LIN {X -0.197,Y -496.201,Z 1484.544,A 0.000,B 0.000,C 90.000,E1 97.936} C_DIS
LIN {X 0.122,Y -496.493,Z 1484.541,A 0.000,B 0.000,C 90.000,E1 97.409} C_DIS
LIN {X -0.111,Y -495.790,Z 1484.539,A 0.000,B 0.000,C 90.000,E1 96.947} C_DIS
LIN {X 0.150,Y -493.977,Z 1484.536,A 0.000,B 0.000,C 90.000,E1 96.429} C_DIS
LIN {X 0.006,Y -492.546,Z 1484.534,A 0.000,B 0.000,C 90.000,E1 96.201} C_DIS
LIN {X -0.163,Y -484.137,Z 1484.528,A 0.000,B 0.000,C 90.000,E1 94.992} C_DIS
LIN {X -0.014,Y -472.049,Z 1484.517,A 0.000,B 0.000,C 90.000,E1 92.980} C_DIS
LIN {X -0.036,Y -464.001,Z 1484.510,A 0.000,B 0.000,C 90.000,E1 91.718} C_DIS
LIN {X 0.053,Y -453.863,Z 1484.501,A 0.000,B 0.000,C 90.000,E1 90.172} C_DIS
LIN {X 0.159,Y -441.677,Z 1484.491,A 0.000,B 0.000,C 90.000,E1 88.339} C_DIS
LIN {X 0.042,Y -429.423,Z 1484.481,A 0.000,B 0.000,C 90.000,E1 86.502} C_DIS
LIN {X -0.173,Y -415.484,Z 1484.469,A 0.000,B 0.000,C 90.000,E1 84.375} C_DIS
LIN {X -0.004,Y -404.925,Z 1484.459,A 0.000,B 0.000,C 90.000,E1 82.704} C_DIS
LIN {X 0.094,Y -392.488,Z 1484.449,A 0.000,B 0.000,C 90.000,E1 80.735} C_DIS
LIN {X 0.042,Y -376.995,Z 1484.434,A 0.000,B 0.000,C 90.000,E1 78.173} C_DIS
LIN {X 0.185,Y -362.226,Z 1484.420,A 0.000,B 0.000,C 90.000,E1 75.519} C_DIS
LIN {X 0.053,Y -350.925,Z 1484.408,A 0.000,B 0.000,C 90.000,E1 73.449} C_DIS
LIN {X -0.007,Y -339.682,Z 1484.396,A 0.000,B 0.000,C 90.000,E1 71.329} C_DIS
LIN {X 0.011,Y -328.550,Z 1484.384,A 0.000,B 0.000,C 90.000,E1 69.156} C_DIS
LIN {X -0.003,Y -311.910,Z 1484.365,A 0.000,B 0.000,C 90.000,E1 65.665} C_DIS
LIN {X -0.046,Y -297.959,Z 1484.347,A 0.000,B 0.000,C 90.000,E1 62.410} C_DIS
LIN {X -0.061,Y -287.479,Z 1484.332,A 0.000,B 0.000,C 90.000,E1 59.744} C_DIS
LIN {X 0.186,Y -276.248,Z 1484.315,A 0.000,B 0.000,C 90.000,E1 56.628} C_DIS
LIN {X -0.025,Y -265.271,Z 1484.297,A 0.000,B 0.000,C 90.000,E1 53.543} C_DIS
LIN {X -0.025,Y -253.773,Z 1484.278,A 0.000,B 0.000,C 90.000,E1 49.989} C_DIS
LIN {X -0.097,Y -243.103,Z 1484.258,A 0.000,B 0.000,C 90.000,E1 46.377} C_DIS
LIN {X 0.079,Y -235.363,Z 1484.241,A 0.000,B 0.000,C 90.000,E1 43.380} C_DIS
LIN {X -0.020,Y -226.608,Z 1484.220,A 0.000,B 0.000,C 90.000,E1 39.644} C_DIS
LIN {X -0.002,Y -220.283,Z 1484.203,A 0.000,B 0.000,C 90.000,E1 36.583} C_DIS
LIN {X 0.007,Y -213.225,Z 1484.182,A 0.000,B 0.000,C 90.000,E1 32.704} C_DIS
LIN {X 0.105,Y -207.137,Z 1484.160,A 0.000,B 0.000,C 90.000,E1 28.743} C_DIS
LIN {X 0.059,Y -201.875,Z 1484.138,A 0.000,B 0.000,C 90.000,E1 24.771} C_DIS
LIN {X 0.031,Y -196.556,Z 1484.111,A 0.000,B 0.000,C 90.000,E1 19.939} C_DIS
LIN {X -0.035,Y -192.268,Z 1484.084,A 0.000,B 0.000,C 90.000,E1 15.064} C_DIS
LIN {X 0.082,Y -188.732,Z 1484.052,A 0.000,B 0.000,C 90.000,E1 9.265} C_DIS
LIN {X -0.046,Y -186.486,Z 1484.019,A 0.000,B 0.000,C 90.000,E1 3.498} C_DIS
LIN {X 0.034,Y -185.763,Z 1483.984,A 0.000,B 0.000,C 90.000,E1 357.020} C_DIS
LIN {X -0.001,Y -186.437,Z 1483.951,A 0.000,B 0.000,C 90.000,E1 351.197} C_DIS
LIN {X -0.087,Y -188.920,Z 1483.914,A 0.000,B 0.000,C 90.000,E1 344.574} C_DIS
LIN {X 0.063,Y -192.234,Z 1483.887,A 0.000,B 0.000,C 90.000,E1 339.571} C_DIS
LIN {X 0.014,Y -195.864,Z 1483.864,A 0.000,B 0.000,C 90.000,E1 335.485} C_DIS
LIN {X -0.045,Y -200.473,Z 1483.841,A 0.000,B 0.000,C 90.000,E1 331.435} C_DIS
LIN {X 0.084,Y -206.120,Z 1483.819,A 0.000,B 0.000,C 90.000,E1 327.375} C_DIS
LIN {X 0.075,Y -211.585,Z 1483.801,A 0.000,B 0.000,C 90.000,E1 324.196} C_DIS
LIN {X -0.068,Y -217.834,Z 1483.784,A 0.000,B 0.000,C 90.000,E1 321.090} C_DIS
LIN {X 0.048,Y -225.078,Z 1483.766,A 0.000,B 0.000,C 90.000,E1 317.957} C_DIS
LIN {X 0.113,Y -234.367,Z 1483.747,A 0.000,B 0.000,C 90.000,E1 314.514} C_DIS
LIN {X 0.146,Y -244.835,Z 1483.729,A 0.000,B 0.000,C 90.000,E1 311.148} C_DIS
LIN {X -0.015,Y -254.072,Z 1483.715,A 0.000,B 0.000,C 90.000,E1 308.624} C_DIS
LIN {X 0.023,Y -263.027,Z 1483.703,A 0.000,B 0.000,C 90.000,E1 306.457} C_DIS
LIN {X 0.002,Y -271.259,Z 1483.693,A 0.000,B 0.000,C 90.000,E1 304.692} C_DIS
LIN {X -0.041,Y -280.539,Z 1483.683,A 0.000,B 0.000,C 90.000,E1 302.959} C_DIS
LIN {X -0.120,Y -292.857,Z 1483.672,A 0.000,B 0.000,C 90.000,E1 300.924} C_DIS
LIN {X 0.122,Y -304.194,Z 1483.662,A 0.000,B 0.000,C 90.000,E1 299.205} C_DIS
LIN {X -0.090,Y -311.599,Z 1483.657,A 0.000,B 0.000,C 90.000,E1 298.281} C_DIS
LIN {X -0.012,Y -327.563,Z 1483.647,A 0.000,B 0.000,C 90.000,E1 296.437} C_DIS
LIN {X -0.040,Y -352.222,Z 1483.633,A 0.000,B 0.000,C 90.000,E1 293.898} C_DIS
LIN {X 0.157,Y -363.050,Z 1483.627,A 0.000,B 0.000,C 90.000,E1 292.770} C_DIS
LIN {X -0.133,Y -373.704,Z 1483.620,A 0.000,B 0.000,C 90.000,E1 291.716} C_DIS
LIN {X -0.119,Y -384.171,Z 1483.614,A 0.000,B 0.000,C 90.000,E1 290.610} C_DIS
LIN {X 0.094,Y -394.100,Z 1483.608,A 0.000,B 0.000,C 90.000,E1 289.504} C_DIS
LIN {X -0.132,Y -403.935,Z 1483.602,A 0.000,B 0.000,C 90.000,E1 288.417} C_DIS
LIN {X -0.156,Y -410.810,Z 1483.598,A 0.000,B 0.000,C 90.000,E1 287.583} C_DIS
LIN {X 0.001,Y -417.219,Z 1483.593,A 0.000,B 0.000,C 90.000,E1 286.732} C_DIS
LIN {X 0.104,Y -422.991,Z 1483.588,A 0.000,B 0.000,C 90.000,E1 285.898} C_DIS
LIN {X 0.144,Y -428.102,Z 1483.584,A 0.000,B 0.000,C 90.000,E1 285.079} C_DIS
LIN {X -0.066,Y -432.329,Z 1483.579,A 0.000,B 0.000,C 90.000,E1 284.300} C_DIS
LIN {X 0.069,Y -435.873,Z 1483.575,A 0.000,B 0.000,C 90.000,E1 283.480} C_DIS
LIN {X 0.139,Y -437.790,Z 1483.572,A 0.000,B 0.000,C 90.000,E1 282.939} C_DIS
LIN {X 0.114,Y -439.351,Z 1483.569,A 0.000,B 0.000,C 90.000,E1 282.411} C_DIS
LIN {X 0.100,Y -440.535,Z 1483.566,A 0.000,B 0.000,C 90.000,E1 281.883} C_DIS
LIN {X 0.006,Y -441.261,Z 1483.563,A 0.000,B 0.000,C 90.000,E1 281.366} C_DIS
LIN {X 0.009,Y -441.485,Z 1483.560,A 0.000,B 0.000,C 90.000,E1 280.838} C_DIS
LIN {X 0.015,Y -441.181,Z 1483.557,A 0.000,B 0.000,C 90.000,E1 280.310} C_DIS
LIN {X -0.057,Y -440.296,Z 1483.554,A 0.000,B 0.000,C 90.000,E1 279.792} C_DIS
LIN {X -0.054,Y -438.823,Z 1483.551,A 0.000,B 0.000,C 90.000,E1 279.265} C_DIS
LIN {X -0.128,Y -436.665,Z 1483.548,A 0.000,B 0.000,C 90.000,E1 278.746} C_DIS
LIN {X -0.144,Y -433.693,Z 1483.546,A 0.000,B 0.000,C 90.000,E1 278.219} C_DIS
LIN {X 0.184,Y -429.791,Z 1483.543,A 0.000,B 0.000,C 90.000,E1 277.644} C_DIS
LIN {X 0.066,Y -424.843,Z 1483.540,A 0.000,B 0.000,C 90.000,E1 277.125} C_DIS
LIN {X 0.036,Y -418.911,Z 1483.537,A 0.000,B 0.000,C 90.000,E1 276.606} C_DIS
LIN {X 0.027,Y -412.593,Z 1483.534,A 0.000,B 0.000,C 90.000,E1 276.144} C_DIS
LIN {X 0.065,Y -406.271,Z 1483.532,A 0.000,B 0.000,C 90.000,E1 275.739} C_DIS
LIN {X -0.003,Y -399.690,Z 1483.530,A 0.000,B 0.000,C 90.000,E1 275.391} C_DIS
LIN {X 0.013,Y -389.854,Z 1483.527,A 0.000,B 0.000,C 90.000,E1 274.935} C_DIS
LIN {X -0.072,Y -374.378,Z 1483.524,A 0.000,B 0.000,C 90.000,E1 274.302} C_DIS
LIN {X 0.041,Y -361.581,Z 1483.521,A 0.000,B 0.000,C 90.000,E1 273.784} C_DIS
LIN {X 0.034,Y -348.652,Z 1483.519,A 0.000,B 0.000,C 90.000,E1 273.326} C_DIS
LIN {X -0.080,Y -338.477,Z 1483.517,A 0.000,B 0.000,C 90.000,E1 273.037} C_DIS
LIN {X -0.048,Y -324.878,Z 1483.515,A 0.000,B 0.000,C 90.000,E1 272.694} C_DIS
LIN {X 0.022,Y -313.880,Z 1483.514,A 0.000,B 0.000,C 90.000,E1 272.465} C_DIS
LIN {X -0.011,Y -300.345,Z 1483.513,A 0.000,B 0.000,C 90.000,E1 272.293} C_DIS
LIN {X -0.077,Y -289.823,Z 1483.512,A 0.000,B 0.000,C 90.000,E1 272.236} C_DIS
LIN {X -0.124,Y -286.503,Z 1483.512,A 0.000,B 0.000,C 90.000,E1 272.236} C_DIS
LIN {X 0.072,Y -181.230,Z 1483.512,A 0.000,B 0.000,C 90.000,E1 272.178} C_DIS
LIN {X 0.063,Y -181.568,Z 1483.503,A 0.000,B 0.000,C 90.000,E1 270.458} C_DIS
LIN {X 0.053,Y -181.117,Z 1483.489,A 0.000,B 0.000,C 90.000,E1 267.936} C_DIS
LIN {X 0.041,Y -180.906,Z 1483.475,A 0.000,B 0.000,C 90.000,E1 265.412} C_DIS
LIN {X -0.083,Y -180.716,Z 1483.470,A 0.000,B 0.000,C 90.000,E1 264.609} C_DIS
LIN {X 0.015,Y -178.803,Z 1483.442,A 0.000,B 0.000,C 90.000,E1 259.511} C_DIS
LIN {X 0.091,Y -175.849,Z 1483.413,A 0.000,B 0.000,C 90.000,E1 254.393} C_DIS
LIN {X 0.051,Y -172.584,Z 1483.390,A 0.000,B 0.000,C 90.000,E1 250.134} C_DIS
LIN {X 0.067,Y -171.473,Z 1483.380,A 0.000,B 0.000,C 90.000,E1 248.411} C_DIS
LIN {X 0.047,Y -167.704,Z 1483.356,A 0.000,B 0.000,C 90.000,E1 244.101} C_DIS
LIN {X 0.060,Y -166.390,Z 1483.347,A 0.000,B 0.000,C 90.000,E1 242.359} C_DIS
LIN {X 0.051,Y -163.117,Z 1483.327,A 0.000,B 0.000,C 90.000,E1 238.869} C_DIS
LIN {X 0.101,Y -161.067,Z 1483.313,A 0.000,B 0.000,C 90.000,E1 236.215} C_DIS
LIN {X -0.012,Y -157.800,Z 1483.293,A 0.000,B 0.000,C 90.000,E1 232.718} C_DIS
LIN {X -0.073,Y -155.836,Z 1483.278,A 0.000,B 0.000,C 90.000,E1 230.070} C_DIS
LIN {X -0.017,Y -152.086,Z 1483.253,A 0.000,B 0.000,C 90.000,E1 225.567} C_DIS
LIN {X 0.002,Y -150.336,Z 1483.238,A 0.000,B 0.000,C 90.000,E1 222.852} C_DIS
LIN {X 0.023,Y -147.076,Z 1483.213,A 0.000,B 0.000,C 90.000,E1 218.302} C_DIS
LIN {X -0.073,Y -145.650,Z 1483.198,A 0.000,B 0.000,C 90.000,E1 215.598} C_DIS
LIN {X -0.068,Y -143.032,Z 1483.172,A 0.000,B 0.000,C 90.000,E1 211.003} C_DIS
LIN {X 0.058,Y -141.657,Z 1483.152,A 0.000,B 0.000,C 90.000,E1 207.257} C_DIS
LIN {X -0.023,Y -139.446,Z 1483.115,A 0.000,B 0.000,C 90.000,E1 200.791} C_DIS
LIN {X 0.030,Y -139.180,Z 1483.105,A 0.000,B 0.000,C 90.000,E1 198.906} C_DIS
LIN {X 0.058,Y -138.320,Z 1483.053,A 0.000,B 0.000,C 90.000,E1 189.557} C_DIS
LIN {X 0.067,Y -139.465,Z 1483.006,A 0.000,B 0.000,C 90.000,E1 181.146} C_DIS
LIN {X 0.009,Y -141.029,Z 1482.975,A 0.000,B 0.000,C 90.000,E1 175.584} C_DIS
LIN {X -0.037,Y -142.396,Z 1482.960,A 0.000,B 0.000,C 90.000,E1 172.818} C_DIS
LIN {X 0.025,Y -144.628,Z 1482.934,A 0.000,B 0.000,C 90.000,E1 168.173} C_DIS
LIN {X -0.057,Y -147.823,Z 1482.909,A 0.000,B 0.000,C 90.000,E1 163.614} C_DIS
LIN {X 0.031,Y -150.514,Z 1482.889,A 0.000,B 0.000,C 90.000,E1 159.934} C_DIS
LIN {X 0.050,Y -153.976,Z 1482.868,A 0.000,B 0.000,C 90.000,E1 156.305} C_DIS
LIN {X -0.028,Y -157.388,Z 1482.849,A 0.000,B 0.000,C 90.000,E1 152.743} C_DIS
LIN {X -0.087,Y -161.592,Z 1482.829,A 0.000,B 0.000,C 90.000,E1 149.203} C_DIS
LIN {X -0.076,Y -165.788,Z 1482.809,A 0.000,B 0.000,C 90.000,E1 145.674} C_DIS
LIN {X -0.091,Y -170.751,Z 1482.790,A 0.000,B 0.000,C 90.000,E1 142.190} C_DIS
LIN {X 0.067,Y -175.623,Z 1482.771,A 0.000,B 0.000,C 90.000,E1 138.690} C_DIS
LIN {X -0.063,Y -181.239,Z 1482.752,A 0.000,B 0.000,C 90.000,E1 135.324} C_DIS
LIN {X 0.067,Y -186.708,Z 1482.733,A 0.000,B 0.000,C 90.000,E1 131.919} C_DIS
LIN {X 0.019,Y -191.308,Z 1482.719,A 0.000,B 0.000,C 90.000,E1 129.439} C_DIS
LIN {X -0.050,Y -197.137,Z 1482.701,A 0.000,B 0.000,C 90.000,E1 126.171} C_DIS
LIN {X -0.035,Y -201.174,Z 1482.689,A 0.000,B 0.000,C 90.000,E1 124.119} C_DIS
LIN {X -0.001,Y -201.373,Z 1482.689,A 0.000,B 0.000,C 90.000,E1 123.992} C_DIS
LIN {X -0.046,Y -314.503,Z 1482.689,A 0.000,B 0.000,C 90.000,E1 123.992} C_DIS
LIN {X -0.172,Y -315.934,Z 1482.689,A 0.000,B 0.000,C 90.000,E1 123.992} C_DIS
LIN {X 0.069,Y -321.100,Z 1482.687,A 0.000,B 0.000,C 90.000,E1 123.706} C_DIS
LIN {X 0.043,Y -324.274,Z 1482.686,A 0.000,B 0.000,C 90.000,E1 123.420} C_DIS
LIN {X 0.155,Y -327.904,Z 1482.683,A 0.000,B 0.000,C 90.000,E1 122.880} C_DIS
LIN {X -0.025,Y -329.447,Z 1482.681,A 0.000,B 0.000,C 90.000,E1 122.594} C_DIS
LIN {X 0.010,Y -342.874,Z 1482.662,A 0.000,B 0.000,C 90.000,E1 119.155} C_DIS
LIN {X -0.017,Y -355.319,Z 1482.647,A 0.000,B 0.000,C 90.000,E1 116.411} C_DIS
LIN {X 0.144,Y -369.261,Z 1482.632,A 0.000,B 0.000,C 90.000,E1 113.695} C_DIS
LIN {X -0.205,Y -383.004,Z 1482.619,A 0.000,B 0.000,C 90.000,E1 111.408} C_DIS
LIN {X 0.007,Y -398.116,Z 1482.606,A 0.000,B 0.000,C 90.000,E1 109.087} C_DIS
LIN {X -0.036,Y -414.704,Z 1482.594,A 0.000,B 0.000,C 90.000,E1 106.858} C_DIS
LIN {X 0.100,Y -432.882,Z 1482.582,A 0.000,B 0.000,C 90.000,E1 104.662} C_DIS
LIN {X -0.096,Y -452.544,Z 1482.570,A 0.000,B 0.000,C 90.000,E1 102.591} C_DIS
LIN {X -0.093,Y -472.851,Z 1482.559,A 0.000,B 0.000,C 90.000,E1 100.658} C_DIS
LIN {X -0.172,Y -488.418,Z 1482.552,A 0.000,B 0.000,C 90.000,E1 99.321} C_DIS
LIN {X -0.094,Y -490.656,Z 1482.550,A 0.000,B 0.000,C 90.000,E1 99.095} C_DIS
LIN {X 0.061,Y -492.347,Z 1482.549,A 0.000,B 0.000,C 90.000,E1 98.859} C_DIS
LIN {X -0.034,Y -493.807,Z 1482.548,A 0.000,B 0.000,C 90.000,E1 98.624} C_DIS
LIN {X -0.202,Y -494.892,Z 1482.547,A 0.000,B 0.000,C 90.000,E1 98.398} C_DIS
LIN {X 0.114,Y -496.149,Z 1482.544,A 0.000,B 0.000,C 90.000,E1 97.871} C_DIS
LIN {X -0.127,Y -496.370,Z 1482.541,A 0.000,B 0.000,C 90.000,E1 97.409} C_DIS
LIN {X 0.132,Y -495.595,Z 1482.538,A 0.000,B 0.000,C 90.000,E1 96.891} C_DIS
LIN {X -0.099,Y -493.693,Z 1482.536,A 0.000,B 0.000,C 90.000,E1 96.429} C_DIS
LIN {X -0.242,Y -492.203,Z 1482.534,A 0.000,B 0.000,C 90.000,E1 96.201} C_DIS
LIN {X 0.070,Y -483.811,Z 1482.527,A 0.000,B 0.000,C 90.000,E1 94.935} C_DIS
LIN {X 0.207,Y -471.696,Z 1482.516,A 0.000,B 0.000,C 90.000,E1 92.922} C_DIS
LIN {X 0.177,Y -463.645,Z 1482.509,A 0.000,B 0.000,C 90.000,E1 91.661} C_DIS
LIN {X -0.197,Y -453.496,Z 1482.501,A 0.000,B 0.000,C 90.000,E1 90.172} C_DIS
LIN {X 0.101,Y -439.614,Z 1482.489,A 0.000,B 0.000,C 90.000,E1 88.051} C_DIS
LIN {X -0.067,Y -427.391,Z 1482.479,A 0.000,B 0.000,C 90.000,E1 86.216} C_DIS
LIN {X -0.008,Y -415.232,Z 1482.468,A 0.000,B 0.000,C 90.000,E1 84.318} C_DIS
LIN {X 0.152,Y -404.703,Z 1482.459,A 0.000,B 0.000,C 90.000,E1 82.648} C_DIS
LIN {X -0.150,Y -392.292,Z 1482.448,A 0.000,B 0.000,C 90.000,E1 80.735} C_DIS
LIN {X -0.198,Y -376.851,Z 1482.434,A 0.000,B 0.000,C 90.000,E1 78.173} C_DIS
LIN {X -0.048,Y -362.083,Z 1482.420,A 0.000,B 0.000,C 90.000,E1 75.519} C_DIS
LIN {X -0.077,Y -350.793,Z 1482.408,A 0.000,B 0.000,C 90.000,E1 73.433} C_DIS
LIN {X 0.090,Y -339.540,Z 1482.396,A 0.000,B 0.000,C 90.000,E1 71.275} C_DIS
LIN {X -0.092,Y -328.391,Z 1482.384,A 0.000,B 0.000,C 90.000,E1 69.135} C_DIS
LIN {X 0.067,Y -311.746,Z 1482.365,A 0.000,B 0.000,C 90.000,E1 65.613} C_DIS
LIN {X 0.009,Y -297.800,Z 1482.346,A 0.000,B 0.000,C 90.000,E1 62.359} C_DIS
LIN {X 0.107,Y -286.054,Z 1482.330,A 0.000,B 0.000,C 90.000,E1 59.331} C_DIS
LIN {X -0.015,Y -276.142,Z 1482.315,A 0.000,B 0.000,C 90.000,E1 56.628} C_DIS
LIN {X 0.076,Y -266.397,Z 1482.299,A 0.000,B 0.000,C 90.000,E1 53.829} C_DIS
LIN {X 0.107,Y -254.835,Z 1482.279,A 0.000,B 0.000,C 90.000,E1 50.275} C_DIS
LIN {X -0.104,Y -245.127,Z 1482.261,A 0.000,B 0.000,C 90.000,E1 47.067} C_DIS
LIN {X -0.040,Y -237.225,Z 1482.245,A 0.000,B 0.000,C 90.000,E1 44.109} C_DIS
LIN {X -0.097,Y -228.340,Z 1482.224,A 0.000,B 0.000,C 90.000,E1 40.378} C_DIS
LIN {X -0.035,Y -221.856,Z 1482.207,A 0.000,B 0.000,C 90.000,E1 37.317} C_DIS
LIN {X -0.028,Y -214.705,Z 1482.186,A 0.000,B 0.000,C 90.000,E1 33.452} C_DIS
LIN {X -0.060,Y -208.438,Z 1482.164,A 0.000,B 0.000,C 90.000,E1 29.539} C_DIS
LIN {X 0.033,Y -203.062,Z 1482.142,A 0.000,B 0.000,C 90.000,E1 25.540} C_DIS
LIN {X -0.018,Y -198.447,Z 1482.120,A 0.000,B 0.000,C 90.000,E1 21.535} C_DIS
LIN {X -0.074,Y -193.824,Z 1482.093,A 0.000,B 0.000,C 90.000,E1 16.677} C_DIS
LIN {X 0.063,Y -190.333,Z 1482.065,A 0.000,B 0.000,C 90.000,E1 11.715} C_DIS
LIN {X -0.067,Y -187.547,Z 1482.033,A 0.000,B 0.000,C 90.000,E1 5.967} C_DIS
LIN {X 0.051,Y -186.066,Z 1481.993,A 0.000,B 0.000,C 90.000,E1 358.682} C_DIS
LIN {X -0.026,Y -186.346,Z 1481.960,A 0.000,B 0.000,C 90.000,E1 352.875} C_DIS
LIN {X -0.054,Y -187.991,Z 1481.928,A 0.000,B 0.000,C 90.000,E1 347.061} C_DIS
LIN {X -0.087,Y -191.206,Z 1481.896,A 0.000,B 0.000,C 90.000,E1 341.275} C_DIS
LIN {X 0.047,Y -195.244,Z 1481.868,A 0.000,B 0.000,C 90.000,E1 336.305} C_DIS
LIN {X 0.054,Y -199.627,Z 1481.846,A 0.000,B 0.000,C 90.000,E1 332.231} C_DIS
LIN {X 0.048,Y -205.025,Z 1481.823,A 0.000,B 0.000,C 90.000,E1 328.201} C_DIS
LIN {X 0.008,Y -210.284,Z 1481.806,A 0.000,B 0.000,C 90.000,E1 325.022} C_DIS
LIN {X -0.124,Y -216.327,Z 1481.788,A 0.000,B 0.000,C 90.000,E1 321.904} C_DIS
LIN {X -0.048,Y -223.331,Z 1481.771,A 0.000,B 0.000,C 90.000,E1 318.771} C_DIS
LIN {X -0.141,Y -231.303,Z 1481.754,A 0.000,B 0.000,C 90.000,E1 315.729} C_DIS
LIN {X -0.039,Y -241.369,Z 1481.735,A 0.000,B 0.000,C 90.000,E1 312.324} C_DIS
LIN {X 0.035,Y -248.831,Z 1481.723,A 0.000,B 0.000,C 90.000,E1 310.092} C_DIS
LIN {X -0.076,Y -257.124,Z 1481.711,A 0.000,B 0.000,C 90.000,E1 307.935} C_DIS
LIN {X -0.145,Y -266.383,Z 1481.699,A 0.000,B 0.000,C 90.000,E1 305.804} C_DIS
LIN {X 0.029,Y -273.154,Z 1481.691,A 0.000,B 0.000,C 90.000,E1 304.358} C_DIS
LIN {X 0.015,Y -282.589,Z 1481.681,A 0.000,B 0.000,C 90.000,E1 302.625} C_DIS
LIN {X -0.028,Y -297.247,Z 1481.668,A 0.000,B 0.000,C 90.000,E1 300.256} C_DIS
LIN {X -0.115,Y -306.561,Z 1481.661,A 0.000,B 0.000,C 90.000,E1 298.949} C_DIS
LIN {X -0.135,Y -314.339,Z 1481.655,A 0.000,B 0.000,C 90.000,E1 297.975} C_DIS
LIN {X -0.015,Y -333.246,Z 1481.644,A 0.000,B 0.000,C 90.000,E1 295.848} C_DIS
LIN {X 0.040,Y -352.274,Z 1481.633,A 0.000,B 0.000,C 90.000,E1 293.898} C_DIS
LIN {X -0.009,Y -362.988,Z 1481.627,A 0.000,B 0.000,C 90.000,E1 292.823} C_DIS
LIN {X -0.075,Y -376.275,Z 1481.619,A 0.000,B 0.000,C 90.000,E1 291.461} C_DIS
LIN {X 0.064,Y -389.204,Z 1481.612,A 0.000,B 0.000,C 90.000,E1 290.066} C_DIS
LIN {X 0.163,Y -396.749,Z 1481.607,A 0.000,B 0.000,C 90.000,E1 289.214} C_DIS
LIN {X -0.042,Y -406.456,Z 1481.601,A 0.000,B 0.000,C 90.000,E1 288.127} C_DIS
LIN {X 0.085,Y -413.192,Z 1481.596,A 0.000,B 0.000,C 90.000,E1 287.275} C_DIS
LIN {X 0.153,Y -419.463,Z 1481.591,A 0.000,B 0.000,C 90.000,E1 286.441} C_DIS
LIN {X -0.135,Y -425.055,Z 1481.587,A 0.000,B 0.000,C 90.000,E1 285.662} C_DIS
LIN {X -0.239,Y -428.397,Z 1481.584,A 0.000,B 0.000,C 90.000,E1 285.134} C_DIS
LIN {X -0.031,Y -432.655,Z 1481.579,A 0.000,B 0.000,C 90.000,E1 284.300} C_DIS
LIN {X 0.107,Y -436.190,Z 1481.575,A 0.000,B 0.000,C 90.000,E1 283.480} C_DIS
LIN {X 0.179,Y -438.099,Z 1481.572,A 0.000,B 0.000,C 90.000,E1 282.939} C_DIS
LIN {X 0.155,Y -439.678,Z 1481.569,A 0.000,B 0.000,C 90.000,E1 282.411} C_DIS
LIN {X 0.142,Y -440.886,Z 1481.566,A 0.000,B 0.000,C 90.000,E1 281.883} C_DIS
LIN {X 0.052,Y -441.623,Z 1481.563,A 0.000,B 0.000,C 90.000,E1 281.366} C_DIS
LIN {X 0.057,Y -441.885,Z 1481.560,A 0.000,B 0.000,C 90.000,E1 280.838} C_DIS
LIN {X 0.064,Y -441.638,Z 1481.557,A 0.000,B 0.000,C 90.000,E1 280.310} C_DIS
LIN {X -0.006,Y -440.799,Z 1481.554,A 0.000,B 0.000,C 90.000,E1 279.792} C_DIS
LIN {X 0.000,Y -439.363,Z 1481.552,A 0.000,B 0.000,C 90.000,E1 279.265} C_DIS
LIN {X -0.072,Y -437.236,Z 1481.549,A 0.000,B 0.000,C 90.000,E1 278.746} C_DIS
LIN {X -0.085,Y -434.334,Z 1481.546,A 0.000,B 0.000,C 90.000,E1 278.219} C_DIS
LIN {X -0.180,Y -430.506,Z 1481.543,A 0.000,B 0.000,C 90.000,E1 277.701} C_DIS
LIN {X 0.132,Y -425.600,Z 1481.540,A 0.000,B 0.000,C 90.000,E1 277.125} C_DIS
LIN {X 0.081,Y -419.682,Z 1481.537,A 0.000,B 0.000,C 90.000,E1 276.606} C_DIS
LIN {X 0.103,Y -413.484,Z 1481.534,A 0.000,B 0.000,C 90.000,E1 276.144} C_DIS
LIN {X 0.096,Y -407.116,Z 1481.532,A 0.000,B 0.000,C 90.000,E1 275.739} C_DIS
LIN {X 0.031,Y -400.572,Z 1481.530,A 0.000,B 0.000,C 90.000,E1 275.391} C_DIS
LIN {X 0.031,Y -390.740,Z 1481.527,A 0.000,B 0.000,C 90.000,E1 274.935} C_DIS
LIN {X -0.099,Y -375.021,Z 1481.524,A 0.000,B 0.000,C 90.000,E1 274.302} C_DIS
LIN {X 0.016,Y -362.205,Z 1481.521,A 0.000,B 0.000,C 90.000,E1 273.784} C_DIS
LIN {X -0.011,Y -352.505,Z 1481.519,A 0.000,B 0.000,C 90.000,E1 273.440} C_DIS
LIN {X 0.132,Y -342.469,Z 1481.517,A 0.000,B 0.000,C 90.000,E1 273.094} C_DIS
LIN {X 0.022,Y -328.689,Z 1481.515,A 0.000,B 0.000,C 90.000,E1 272.751} C_DIS
LIN {X 0.045,Y -317.797,Z 1481.514,A 0.000,B 0.000,C 90.000,E1 272.522} C_DIS
LIN {X -0.046,Y -310.093,Z 1481.513,A 0.000,B 0.000,C 90.000,E1 272.407} C_DIS
LIN {X 0.128,Y -297.244,Z 1481.513,A 0.000,B 0.000,C 90.000,E1 272.236} C_DIS
LIN {X -0.099,Y -287.867,Z 1481.512,A 0.000,B 0.000,C 90.000,E1 272.236} C_DIS
LIN {X 0.088,Y -181.229,Z 1481.512,A 0.000,B 0.000,C 90.000,E1 272.178} C_DIS
LIN {X 0.049,Y -181.568,Z 1481.503,A 0.000,B 0.000,C 90.000,E1 270.458} C_DIS
LIN {X -0.091,Y -181.003,Z 1481.484,A 0.000,B 0.000,C 90.000,E1 267.135} C_DIS
LIN {X 0.026,Y -180.907,Z 1481.475,A 0.000,B 0.000,C 90.000,E1 265.412} C_DIS
LIN {X -0.098,Y -180.714,Z 1481.470,A 0.000,B 0.000,C 90.000,E1 264.609} C_DIS
LIN {X 0.001,Y -178.801,Z 1481.442,A 0.000,B 0.000,C 90.000,E1 259.511} C_DIS
LIN {X 0.078,Y -175.846,Z 1481.413,A 0.000,B 0.000,C 90.000,E1 254.393} C_DIS
LIN {X 0.077,Y -172.038,Z 1481.385,A 0.000,B 0.000,C 90.000,E1 249.263} C_DIS
LIN {X 0.053,Y -171.469,Z 1481.380,A 0.000,B 0.000,C 90.000,E1 248.411} C_DIS
LIN {X 0.033,Y -167.701,Z 1481.356,A 0.000,B 0.000,C 90.000,E1 244.101} C_DIS
LIN {X 0.046,Y -166.386,Z 1481.347,A 0.000,B 0.000,C 90.000,E1 242.359} C_DIS
LIN {X 0.038,Y -163.113,Z 1481.327,A 0.000,B 0.000,C 90.000,E1 238.869} C_DIS
LIN {X 0.088,Y -161.062,Z 1481.313,A 0.000,B 0.000,C 90.000,E1 236.215} C_DIS
LIN {X -0.025,Y -157.796,Z 1481.293,A 0.000,B 0.000,C 90.000,E1 232.718} C_DIS
LIN {X 0.014,Y -155.832,Z 1481.278,A 0.000,B 0.000,C 90.000,E1 230.033} C_DIS
LIN {X -0.029,Y -152.083,Z 1481.253,A 0.000,B 0.000,C 90.000,E1 225.567} C_DIS
LIN {X -0.010,Y -150.333,Z 1481.238,A 0.000,B 0.000,C 90.000,E1 222.852} C_DIS
LIN {X 0.010,Y -147.073,Z 1481.213,A 0.000,B 0.000,C 90.000,E1 218.302} C_DIS
LIN {X -0.086,Y -145.647,Z 1481.198,A 0.000,B 0.000,C 90.000,E1 215.598} C_DIS
LIN {X -0.081,Y -143.030,Z 1481.172,A 0.000,B 0.000,C 90.000,E1 211.003} C_DIS
LIN {X 0.046,Y -141.655,Z 1481.151,A 0.000,B 0.000,C 90.000,E1 207.257} C_DIS
LIN {X -0.035,Y -139.445,Z 1481.115,A 0.000,B 0.000,C 90.000,E1 200.791} C_DIS
LIN {X 0.017,Y -139.179,Z 1481.105,A 0.000,B 0.000,C 90.000,E1 198.906} C_DIS
LIN {X 0.046,Y -138.320,Z 1481.053,A 0.000,B 0.000,C 90.000,E1 189.557} C_DIS
LIN {X 0.055,Y -139.467,Z 1481.006,A 0.000,B 0.000,C 90.000,E1 181.146} C_DIS
LIN {X -0.004,Y -141.032,Z 1480.975,A 0.000,B 0.000,C 90.000,E1 175.584} C_DIS
LIN {X -0.050,Y -142.398,Z 1480.960,A 0.000,B 0.000,C 90.000,E1 172.818} C_DIS
LIN {X 0.013,Y -144.631,Z 1480.934,A 0.000,B 0.000,C 90.000,E1 168.173} C_DIS
LIN {X 0.074,Y -147.826,Z 1480.909,A 0.000,B 0.000,C 90.000,E1 163.559} C_DIS
LIN {X 0.017,Y -150.519,Z 1480.889,A 0.000,B 0.000,C 90.000,E1 159.934} C_DIS
LIN {X 0.038,Y -153.981,Z 1480.868,A 0.000,B 0.000,C 90.000,E1 156.305} C_DIS
LIN {X -0.042,Y -157.393,Z 1480.849,A 0.000,B 0.000,C 90.000,E1 152.743} C_DIS
LIN {X 0.039,Y -161.598,Z 1480.829,A 0.000,B 0.000,C 90.000,E1 149.154} C_DIS
LIN {X -0.089,Y -165.795,Z 1480.809,A 0.000,B 0.000,C 90.000,E1 145.674} C_DIS
LIN {X 0.031,Y -170.758,Z 1480.790,A 0.000,B 0.000,C 90.000,E1 142.145} C_DIS
LIN {X 0.053,Y -175.630,Z 1480.771,A 0.000,B 0.000,C 90.000,E1 138.690} C_DIS
LIN {X -0.078,Y -181.245,Z 1480.752,A 0.000,B 0.000,C 90.000,E1 135.324} C_DIS
LIN {X 0.053,Y -186.716,Z 1480.733,A 0.000,B 0.000,C 90.000,E1 131.919} C_DIS
LIN {X 0.004,Y -191.315,Z 1480.719,A 0.000,B 0.000,C 90.000,E1 129.439} C_DIS
LIN {X -0.065,Y -197.146,Z 1480.701,A 0.000,B 0.000,C 90.000,E1 126.171} C_DIS
LIN {X -0.048,Y -201.180,Z 1480.689,A 0.000,B 0.000,C 90.000,E1 124.119} C_DIS
LIN {X -0.059,Y -201.320,Z 1480.689,A 0.000,B 0.000,C 90.000,E1 124.040} C_DIS
LIN {X 0.120,Y -314.129,Z 1480.689,A 0.000,B 0.000,C 90.000,E1 123.992} C_DIS
LIN {X -0.022,Y -315.844,Z 1480.689,A 0.000,B 0.000,C 90.000,E1 123.992} C_DIS
LIN {X 0.045,Y -321.408,Z 1480.687,A 0.000,B 0.000,C 90.000,E1 123.706} C_DIS
LIN {X -0.057,Y -324.547,Z 1480.686,A 0.000,B 0.000,C 90.000,E1 123.420} C_DIS
LIN {X -0.078,Y -328.148,Z 1480.683,A 0.000,B 0.000,C 90.000,E1 122.880} C_DIS
LIN {X 0.020,Y -329.610,Z 1480.681,A 0.000,B 0.000,C 90.000,E1 122.546} C_DIS
LIN {X 0.090,Y -341.721,Z 1480.663,A 0.000,B 0.000,C 90.000,E1 119.411} C_DIS
LIN {X 0.026,Y -354.030,Z 1480.648,A 0.000,B 0.000,C 90.000,E1 116.668} C_DIS
LIN {X 0.158,Y -367.818,Z 1480.633,A 0.000,B 0.000,C 90.000,E1 113.951} C_DIS
LIN {X -0.081,Y -381.417,Z 1480.620,A 0.000,B 0.000,C 90.000,E1 111.642} C_DIS
LIN {X 0.088,Y -396.374,Z 1480.607,A 0.000,B 0.000,C 90.000,E1 109.322} C_DIS
LIN {X 0.000,Y -412.795,Z 1480.595,A 0.000,B 0.000,C 90.000,E1 107.094} C_DIS
LIN {X 0.085,Y -430.794,Z 1480.583,A 0.000,B 0.000,C 90.000,E1 104.898} C_DIS
LIN {X -0.211,Y -450.327,Z 1480.571,A 0.000,B 0.000,C 90.000,E1 102.827} C_DIS
LIN {X 0.102,Y -470.575,Z 1480.560,A 0.000,B 0.000,C 90.000,E1 100.838} C_DIS
LIN {X 0.068,Y -488.718,Z 1480.552,A 0.000,B 0.000,C 90.000,E1 99.265} C_DIS
LIN {X 0.213,Y -490.861,Z 1480.550,A 0.000,B 0.000,C 90.000,E1 99.029} C_DIS
LIN {X -0.205,Y -492.489,Z 1480.549,A 0.000,B 0.000,C 90.000,E1 98.859} C_DIS
LIN {X 0.189,Y -493.887,Z 1480.548,A 0.000,B 0.000,C 90.000,E1 98.568} C_DIS
LIN {X 0.021,Y -494.919,Z 1480.546,A 0.000,B 0.000,C 90.000,E1 98.341} C_DIS
LIN {X -0.153,Y -496.094,Z 1480.544,A 0.000,B 0.000,C 90.000,E1 97.871} C_DIS
LIN {X 0.098,Y -496.241,Z 1480.541,A 0.000,B 0.000,C 90.000,E1 97.352} C_DIS
LIN {X -0.134,Y -495.388,Z 1480.538,A 0.000,B 0.000,C 90.000,E1 96.891} C_DIS
LIN {X 0.125,Y -493.391,Z 1480.536,A 0.000,B 0.000,C 90.000,E1 96.372} C_DIS
LIN {X -0.111,Y -490.091,Z 1480.533,A 0.000,B 0.000,C 90.000,E1 95.910} C_DIS
LIN {X -0.005,Y -480.369,Z 1480.525,A 0.000,B 0.000,C 90.000,E1 94.416} C_DIS
LIN {X -0.060,Y -471.341,Z 1480.516,A 0.000,B 0.000,C 90.000,E1 92.922} C_DIS
LIN {X 0.100,Y -464.933,Z 1480.511,A 0.000,B 0.000,C 90.000,E1 91.892} C_DIS
LIN {X 0.216,Y -454.837,Z 1480.502,A 0.000,B 0.000,C 90.000,E1 90.344} C_DIS
LIN {X -0.109,Y -442.709,Z 1480.492,A 0.000,B 0.000,C 90.000,E1 88.568} C_DIS
LIN {X -0.192,Y -430.590,Z 1480.482,A 0.000,B 0.000,C 90.000,E1 86.731} C_DIS
LIN {X 0.047,Y -416.699,Z 1480.470,A 0.000,B 0.000,C 90.000,E1 84.546} C_DIS
LIN {X -0.165,Y -406.222,Z 1480.461,A 0.000,B 0.000,C 90.000,E1 82.932} C_DIS
LIN {X -0.095,Y -393.857,Z 1480.450,A 0.000,B 0.000,C 90.000,E1 80.971} C_DIS
LIN {X -0.084,Y -376.687,Z 1480.434,A 0.000,B 0.000,C 90.000,E1 78.117} C_DIS
LIN {X 0.052,Y -361.924,Z 1480.419,A 0.000,B 0.000,C 90.000,E1 75.463} C_DIS
LIN {X 0.015,Y -350.639,Z 1480.408,A 0.000,B 0.000,C 90.000,E1 73.378} C_DIS
LIN {X 0.170,Y -337.787,Z 1480.394,A 0.000,B 0.000,C 90.000,E1 70.913} C_DIS
LIN {X -0.082,Y -325.075,Z 1480.380,A 0.000,B 0.000,C 90.000,E1 68.465} C_DIS
LIN {X 0.167,Y -310.135,Z 1480.363,A 0.000,B 0.000,C 90.000,E1 65.229} C_DIS
LIN {X 0.059,Y -296.295,Z 1480.344,A 0.000,B 0.000,C 90.000,E1 61.975} C_DIS
LIN {X -0.131,Y -284.640,Z 1480.328,A 0.000,B 0.000,C 90.000,E1 58.997} C_DIS
LIN {X 0.100,Y -274.799,Z 1480.312,A 0.000,B 0.000,C 90.000,E1 56.215} C_DIS
LIN {X -0.152,Y -263.943,Z 1480.295,A 0.000,B 0.000,C 90.000,E1 53.130} C_DIS
LIN {X -0.032,Y -252.547,Z 1480.275,A 0.000,B 0.000,C 90.000,E1 49.542} C_DIS
LIN {X -0.133,Y -243.046,Z 1480.257,A 0.000,B 0.000,C 90.000,E1 46.296} C_DIS
LIN {X 0.043,Y -235.358,Z 1480.241,A 0.000,B 0.000,C 90.000,E1 43.299} C_DIS
LIN {X -0.055,Y -226.702,Z 1480.220,A 0.000,B 0.000,C 90.000,E1 39.564} C_DIS
LIN {X -0.035,Y -220.449,Z 1480.203,A 0.000,B 0.000,C 90.000,E1 36.503} C_DIS
LIN {X -0.022,Y -213.503,Z 1480.181,A 0.000,B 0.000,C 90.000,E1 32.625} C_DIS
LIN {X -0.019,Y -207.472,Z 1480.159,A 0.000,B 0.000,C 90.000,E1 28.693} C_DIS
LIN {X -0.046,Y -202.294,Z 1480.137,A 0.000,B 0.000,C 90.000,E1 24.719} C_DIS
LIN {X 0.061,Y -197.809,Z 1480.115,A 0.000,B 0.000,C 90.000,E1 20.663} C_DIS
LIN {X 0.040,Y -193.428,Z 1480.088,A 0.000,B 0.000,C 90.000,E1 15.788} C_DIS
LIN {X -0.068,Y -190.110,Z 1480.060,A 0.000,B 0.000,C 90.000,E1 10.894} C_DIS
LIN {X -0.071,Y -187.508,Z 1480.028,A 0.000,B 0.000,C 90.000,E1 5.106} C_DIS
LIN {X -0.041,Y -186.301,Z 1479.988,A 0.000,B 0.000,C 90.000,E1 357.879} C_DIS
LIN {X 0.031,Y -186.937,Z 1479.951,A 0.000,B 0.000,C 90.000,E1 351.197} C_DIS
LIN {X -0.030,Y -189.372,Z 1479.914,A 0.000,B 0.000,C 90.000,E1 344.574} C_DIS
LIN {X -0.044,Y -192.606,Z 1479.887,A 0.000,B 0.000,C 90.000,E1 339.625} C_DIS
LIN {X -0.079,Y -196.192,Z 1479.864,A 0.000,B 0.000,C 90.000,E1 335.537} C_DIS
LIN {X 0.052,Y -200.760,Z 1479.841,A 0.000,B 0.000,C 90.000,E1 331.435} C_DIS
LIN {X -0.091,Y -206.389,Z 1479.819,A 0.000,B 0.000,C 90.000,E1 327.454} C_DIS
LIN {X -0.102,Y -211.860,Z 1479.801,A 0.000,B 0.000,C 90.000,E1 324.276} C_DIS
LIN {X 0.062,Y -218.110,Z 1479.784,A 0.000,B 0.000,C 90.000,E1 321.090} C_DIS
LIN {X 0.022,Y -225.387,Z 1479.767,A 0.000,B 0.000,C 90.000,E1 318.000} C_DIS
LIN {X -0.063,Y -234.674,Z 1479.748,A 0.000,B 0.000,C 90.000,E1 314.595} C_DIS
LIN {X -0.027,Y -245.156,Z 1479.729,A 0.000,B 0.000,C 90.000,E1 311.229} C_DIS
LIN {X -0.028,Y -254.421,Z 1479.715,A 0.000,B 0.000,C 90.000,E1 308.669} C_DIS
LIN {X 0.011,Y -263.341,Z 1479.703,A 0.000,B 0.000,C 90.000,E1 306.503} C_DIS
LIN {X -0.012,Y -271.489,Z 1479.693,A 0.000,B 0.000,C 90.000,E1 304.739} C_DIS
LIN {X -0.152,Y -278.792,Z 1479.685,A 0.000,B 0.000,C 90.000,E1 303.372} C_DIS
LIN {X 0.132,Y -290.835,Z 1479.674,A 0.000,B 0.000,C 90.000,E1 301.258} C_DIS
LIN {X -0.057,Y -301.788,Z 1479.664,A 0.000,B 0.000,C 90.000,E1 299.617} C_DIS
LIN {X 0.079,Y -311.610,Z 1479.657,A 0.000,B 0.000,C 90.000,E1 298.281} C_DIS
LIN {X -0.141,Y -325.225,Z 1479.648,A 0.000,B 0.000,C 90.000,E1 296.744} C_DIS
LIN {X 0.058,Y -344.186,Z 1479.637,A 0.000,B 0.000,C 90.000,E1 294.719} C_DIS
LIN {X -0.141,Y -357.867,Z 1479.630,A 0.000,B 0.000,C 90.000,E1 293.387} C_DIS
LIN {X 0.029,Y -368.405,Z 1479.624,A 0.000,B 0.000,C 90.000,E1 292.280} C_DIS
LIN {X 0.031,Y -379.046,Z 1479.618,A 0.000,B 0.000,C 90.000,E1 291.173} C_DIS
LIN {X 0.050,Y -389.402,Z 1479.612,A 0.000,B 0.000,C 90.000,E1 290.066} C_DIS
LIN {X -0.033,Y -399.447,Z 1479.605,A 0.000,B 0.000,C 90.000,E1 288.960} C_DIS
LIN {X -0.054,Y -406.661,Z 1479.601,A 0.000,B 0.000,C 90.000,E1 288.127} C_DIS
LIN {X 0.068,Y -413.442,Z 1479.596,A 0.000,B 0.000,C 90.000,E1 287.275} C_DIS
LIN {X 0.137,Y -419.705,Z 1479.591,A 0.000,B 0.000,C 90.000,E1 286.441} C_DIS
LIN {X -0.149,Y -425.348,Z 1479.587,A 0.000,B 0.000,C 90.000,E1 285.662} C_DIS
LIN {X -0.250,Y -428.713,Z 1479.584,A 0.000,B 0.000,C 90.000,E1 285.134} C_DIS
LIN {X -0.041,Y -432.995,Z 1479.579,A 0.000,B 0.000,C 90.000,E1 284.300} C_DIS
LIN {X 0.101,Y -436.505,Z 1479.575,A 0.000,B 0.000,C 90.000,E1 283.480} C_DIS
LIN {X 0.174,Y -438.423,Z 1479.572,A 0.000,B 0.000,C 90.000,E1 282.939} C_DIS
LIN {X 0.153,Y -440.007,Z 1479.569,A 0.000,B 0.000,C 90.000,E1 282.411} C_DIS
LIN {X 0.143,Y -441.267,Z 1479.566,A 0.000,B 0.000,C 90.000,E1 281.883} C_DIS
LIN {X 0.053,Y -442.001,Z 1479.563,A 0.000,B 0.000,C 90.000,E1 281.366} C_DIS
LIN {X 0.061,Y -442.307,Z 1479.560,A 0.000,B 0.000,C 90.000,E1 280.838} C_DIS
LIN {X 0.070,Y -442.030,Z 1479.557,A 0.000,B 0.000,C 90.000,E1 280.310} C_DIS
LIN {X 0.003,Y -441.255,Z 1479.554,A 0.000,B 0.000,C 90.000,E1 279.792} C_DIS
LIN {X 0.010,Y -439.835,Z 1479.552,A 0.000,B 0.000,C 90.000,E1 279.265} C_DIS
LIN {X -0.058,Y -437.759,Z 1479.549,A 0.000,B 0.000,C 90.000,E1 278.746} C_DIS
LIN {X -0.069,Y -434.895,Z 1479.546,A 0.000,B 0.000,C 90.000,E1 278.219} C_DIS
LIN {X -0.161,Y -431.139,Z 1479.543,A 0.000,B 0.000,C 90.000,E1 277.701} C_DIS
LIN {X 0.154,Y -426.304,Z 1479.540,A 0.000,B 0.000,C 90.000,E1 277.125} C_DIS
LIN {X -0.086,Y -423.463,Z 1479.538,A 0.000,B 0.000,C 90.000,E1 276.891} C_DIS
LIN {X 0.085,Y -417.359,Z 1479.536,A 0.000,B 0.000,C 90.000,E1 276.372} C_DIS
LIN {X -0.105,Y -411.070,Z 1479.533,A 0.000,B 0.000,C 90.000,E1 275.967} C_DIS
LIN {X 0.009,Y -404.620,Z 1479.531,A 0.000,B 0.000,C 90.000,E1 275.568} C_DIS
LIN {X 0.069,Y -397.982,Z 1479.529,A 0.000,B 0.000,C 90.000,E1 275.220} C_DIS
LIN {X -0.166,Y -388.122,Z 1479.527,A 0.000,B 0.000,C 90.000,E1 274.816} C_DIS
LIN {X 0.152,Y -372.402,Z 1479.523,A 0.000,B 0.000,C 90.000,E1 274.131} C_DIS
LIN {X -0.017,Y -359.774,Z 1479.520,A 0.000,B 0.000,C 90.000,E1 273.669} C_DIS
LIN {X 0.075,Y -346.702,Z 1479.518,A 0.000,B 0.000,C 90.000,E1 273.212} C_DIS
LIN {X 0.046,Y -336.434,Z 1479.516,A 0.000,B 0.000,C 90.000,E1 272.922} C_DIS
LIN {X -0.059,Y -326.270,Z 1479.515,A 0.000,B 0.000,C 90.000,E1 272.694} C_DIS
LIN {X 0.014,Y -314.935,Z 1479.514,A 0.000,B 0.000,C 90.000,E1 272.465} C_DIS
LIN {X -0.028,Y -306.599,Z 1479.513,A 0.000,B 0.000,C 90.000,E1 272.350} C_DIS
LIN {X -0.147,Y -298.533,Z 1479.513,A 0.000,B 0.000,C 90.000,E1 272.293} C_DIS
LIN {X -0.121,Y -285.828,Z 1479.512,A 0.000,B 0.000,C 90.000,E1 272.236} C_DIS
LIN {X 0.076,Y -181.230,Z 1479.512,A 0.000,B 0.000,C 90.000,E1 272.178} C_DIS
LIN {X 0.077,Y -181.567,Z 1479.503,A 0.000,B 0.000,C 90.000,E1 270.458} C_DIS
LIN {X 0.066,Y -181.117,Z 1479.489,A 0.000,B 0.000,C 90.000,E1 267.936} C_DIS
LIN {X 0.054,Y -180.906,Z 1479.475,A 0.000,B 0.000,C 90.000,E1 265.412} C_DIS
LIN {X -0.070,Y -180.718,Z 1479.470,A 0.000,B 0.000,C 90.000,E1 264.609} C_DIS
LIN {X 0.028,Y -178.806,Z 1479.442,A 0.000,B 0.000,C 90.000,E1 259.511} C_DIS
LIN {X -0.065,Y -175.851,Z 1479.413,A 0.000,B 0.000,C 90.000,E1 254.448} C_DIS
LIN {X -0.082,Y -173.177,Z 1479.395,A 0.000,B 0.000,C 90.000,E1 251.040} C_DIS
LIN {X 0.080,Y -171.477,Z 1479.380,A 0.000,B 0.000,C 90.000,E1 248.411} C_DIS
LIN {X -0.091,Y -167.707,Z 1479.356,A 0.000,B 0.000,C 90.000,E1 244.152} C_DIS
LIN {X 0.072,Y -166.395,Z 1479.347,A 0.000,B 0.000,C 90.000,E1 242.359} C_DIS
LIN {X 0.063,Y -163.120,Z 1479.327,A 0.000,B 0.000,C 90.000,E1 238.869} C_DIS
LIN {X -0.110,Y -161.071,Z 1479.313,A 0.000,B 0.000,C 90.000,E1 236.294} C_DIS
LIN {X 0.000,Y -157.803,Z 1479.293,A 0.000,B 0.000,C 90.000,E1 232.718} C_DIS
LIN {X -0.061,Y -155.839,Z 1479.278,A 0.000,B 0.000,C 90.000,E1 230.070} C_DIS
LIN {X -0.005,Y -152.089,Z 1479.253,A 0.000,B 0.000,C 90.000,E1 225.567} C_DIS
LIN {X 0.014,Y -150.340,Z 1479.238,A 0.000,B 0.000,C 90.000,E1 222.852} C_DIS
LIN {X 0.034,Y -147.078,Z 1479.213,A 0.000,B 0.000,C 90.000,E1 218.302} C_DIS
LIN {X -0.062,Y -145.652,Z 1479.198,A 0.000,B 0.000,C 90.000,E1 215.598} C_DIS
LIN {X -0.058,Y -143.034,Z 1479.172,A 0.000,B 0.000,C 90.000,E1 211.003} C_DIS
LIN {X 0.069,Y -141.659,Z 1479.152,A 0.000,B 0.000,C 90.000,E1 207.257} C_DIS
LIN {X -0.011,Y -139.447,Z 1479.115,A 0.000,B 0.000,C 90.000,E1 200.791} C_DIS
LIN {X 0.041,Y -139.181,Z 1479.105,A 0.000,B 0.000,C 90.000,E1 198.906} C_DIS
LIN {X -0.067,Y -138.320,Z 1479.053,A 0.000,B 0.000,C 90.000,E1 189.613} C_DIS
LIN {X -0.061,Y -139.464,Z 1479.007,A 0.000,B 0.000,C 90.000,E1 181.203} C_DIS
LIN {X 0.019,Y -141.027,Z 1478.975,A 0.000,B 0.000,C 90.000,E1 175.584} C_DIS
LIN {X -0.026,Y -142.393,Z 1478.960,A 0.000,B 0.000,C 90.000,E1 172.818} C_DIS
LIN {X 0.036,Y -144.625,Z 1478.934,A 0.000,B 0.000,C 90.000,E1 168.173} C_DIS
LIN {X -0.045,Y -147.820,Z 1478.909,A 0.000,B 0.000,C 90.000,E1 163.614} C_DIS
LIN {X 0.042,Y -150.511,Z 1478.889,A 0.000,B 0.000,C 90.000,E1 159.934} C_DIS
LIN {X -0.079,Y -153.971,Z 1478.869,A 0.000,B 0.000,C 90.000,E1 156.357} C_DIS
LIN {X -0.016,Y -157.383,Z 1478.849,A 0.000,B 0.000,C 90.000,E1 152.743} C_DIS
LIN {X -0.074,Y -161.586,Z 1478.829,A 0.000,B 0.000,C 90.000,E1 149.203} C_DIS
LIN {X -0.063,Y -165.784,Z 1478.809,A 0.000,B 0.000,C 90.000,E1 145.674} C_DIS
LIN {X -0.078,Y -170.744,Z 1478.790,A 0.000,B 0.000,C 90.000,E1 142.190} C_DIS
LIN {X 0.080,Y -175.616,Z 1478.771,A 0.000,B 0.000,C 90.000,E1 138.690} C_DIS
LIN {X -0.050,Y -181.233,Z 1478.752,A 0.000,B 0.000,C 90.000,E1 135.324} C_DIS
LIN {X 0.081,Y -186.701,Z 1478.733,A 0.000,B 0.000,C 90.000,E1 131.919} C_DIS
LIN {X 0.032,Y -191.301,Z 1478.719,A 0.000,B 0.000,C 90.000,E1 129.439} C_DIS
LIN {X -0.036,Y -197.130,Z 1478.701,A 0.000,B 0.000,C 90.000,E1 126.171} C_DIS
LIN {X -0.018,Y -201.164,Z 1478.690,A 0.000,B 0.000,C 90.000,E1 124.119} C_DIS
LIN {X 0.040,Y -201.272,Z 1478.689,A 0.000,B 0.000,C 90.000,E1 124.040} C_DIS
LIN {X 0.009,Y -314.191,Z 1478.689,A 0.000,B 0.000,C 90.000,E1 124.040} C_DIS
LIN {X 0.066,Y -319.275,Z 1478.688,A 0.000,B 0.000,C 90.000,E1 123.865} C_DIS
LIN {X 0.091,Y -321.541,Z 1478.687,A 0.000,B 0.000,C 90.000,E1 123.706} C_DIS
LIN {X 0.123,Y -325.408,Z 1478.685,A 0.000,B 0.000,C 90.000,E1 123.293} C_DIS
LIN {X -0.078,Y -327.310,Z 1478.683,A 0.000,B 0.000,C 90.000,E1 123.038} C_DIS
LIN {X -0.101,Y -328.806,Z 1478.682,A 0.000,B 0.000,C 90.000,E1 122.752} C_DIS
LIN {X 0.068,Y -333.565,Z 1478.675,A 0.000,B 0.000,C 90.000,E1 121.465} C_DIS
LIN {X -0.054,Y -344.854,Z 1478.659,A 0.000,B 0.000,C 90.000,E1 118.693} C_DIS
LIN {X 0.125,Y -357.548,Z 1478.644,A 0.000,B 0.000,C 90.000,E1 115.924} C_DIS
LIN {X 0.034,Y -371.752,Z 1478.629,A 0.000,B 0.000,C 90.000,E1 113.259} C_DIS
LIN {X 0.101,Y -385.749,Z 1478.616,A 0.000,B 0.000,C 90.000,E1 110.918} C_DIS
LIN {X -0.113,Y -401.136,Z 1478.604,A 0.000,B 0.000,C 90.000,E1 108.671} C_DIS
LIN {X -0.081,Y -418.019,Z 1478.591,A 0.000,B 0.000,C 90.000,E1 106.441} C_DIS
LIN {X 0.136,Y -436.517,Z 1478.579,A 0.000,B 0.000,C 90.000,E1 104.245} C_DIS
LIN {X 0.071,Y -456.337,Z 1478.568,A 0.000,B 0.000,C 90.000,E1 102.187} C_DIS
LIN {X -0.128,Y -476.747,Z 1478.557,A 0.000,B 0.000,C 90.000,E1 100.310} C_DIS
LIN {X -0.206,Y -489.620,Z 1478.551,A 0.000,B 0.000,C 90.000,E1 99.208} C_DIS
LIN {X -0.121,Y -491.566,Z 1478.550,A 0.000,B 0.000,C 90.000,E1 98.973} C_DIS
LIN {X -0.113,Y -493.050,Z 1478.548,A 0.000,B 0.000,C 90.000,E1 98.746} C_DIS
LIN {X -0.205,Y -494.276,Z 1478.547,A 0.000,B 0.000,C 90.000,E1 98.511} C_DIS
LIN {X 0.191,Y -495.168,Z 1478.546,A 0.000,B 0.000,C 90.000,E1 98.219} C_DIS
LIN {X -0.052,Y -496.105,Z 1478.543,A 0.000,B 0.000,C 90.000,E1 97.757} C_DIS
LIN {X 0.202,Y -496.035,Z 1478.540,A 0.000,B 0.000,C 90.000,E1 97.239} C_DIS
LIN {X -0.029,Y -494.951,Z 1478.538,A 0.000,B 0.000,C 90.000,E1 96.777} C_DIS
LIN {X -0.117,Y -493.978,Z 1478.536,A 0.000,B 0.000,C 90.000,E1 96.543} C_DIS
LIN {X 0.229,Y -492.656,Z 1478.535,A 0.000,B 0.000,C 90.000,E1 96.258} C_DIS
LIN {X -0.107,Y -482.666,Z 1478.527,A 0.000,B 0.000,C 90.000,E1 94.821} C_DIS
LIN {X 0.195,Y -472.075,Z 1478.517,A 0.000,B 0.000,C 90.000,E1 93.037} C_DIS
LIN {X 0.175,Y -464.095,Z 1478.510,A 0.000,B 0.000,C 90.000,E1 91.776} C_DIS
LIN {X -0.194,Y -453.970,Z 1478.501,A 0.000,B 0.000,C 90.000,E1 90.286} C_DIS
LIN {X 0.116,Y -440.133,Z 1478.490,A 0.000,B 0.000,C 90.000,E1 88.165} C_DIS
LIN {X -0.045,Y -428.036,Z 1478.480,A 0.000,B 0.000,C 90.000,E1 86.331} C_DIS
LIN {X 0.033,Y -415.926,Z 1478.469,A 0.000,B 0.000,C 90.000,E1 84.432} C_DIS
LIN {X -0.194,Y -405.475,Z 1478.460,A 0.000,B 0.000,C 90.000,E1 82.818} C_DIS
LIN {X -0.082,Y -393.132,Z 1478.449,A 0.000,B 0.000,C 90.000,E1 80.849} C_DIS
LIN {X -0.080,Y -376.040,Z 1478.433,A 0.000,B 0.000,C 90.000,E1 77.993} C_DIS
LIN {X 0.048,Y -361.295,Z 1478.419,A 0.000,B 0.000,C 90.000,E1 75.338} C_DIS
LIN {X -0.098,Y -350.000,Z 1478.407,A 0.000,B 0.000,C 90.000,E1 73.268} C_DIS
LIN {X 0.149,Y -337.169,Z 1478.393,A 0.000,B 0.000,C 90.000,E1 70.786} C_DIS
LIN {X 0.149,Y -322.924,Z 1478.378,A 0.000,B 0.000,C 90.000,E1 67.975} C_DIS
LIN {X 0.036,Y -308.132,Z 1478.360,A 0.000,B 0.000,C 90.000,E1 64.793} C_DIS
LIN {X 0.005,Y -294.427,Z 1478.342,A 0.000,B 0.000,C 90.000,E1 61.513} C_DIS
LIN {X 0.125,Y -281.653,Z 1478.323,A 0.000,B 0.000,C 90.000,E1 58.122} C_DIS
LIN {X -0.049,Y -273.086,Z 1478.310,A 0.000,B 0.000,C 90.000,E1 55.754} C_DIS
LIN {X -0.030,Y -262.355,Z 1478.292,A 0.000,B 0.000,C 90.000,E1 52.603} C_DIS
LIN {X 0.039,Y -251.075,Z 1478.272,A 0.000,B 0.000,C 90.000,E1 49.013} C_DIS
LIN {X -0.114,Y -240.760,Z 1478.252,A 0.000,B 0.000,C 90.000,E1 45.405} C_DIS
LIN {X 0.014,Y -233.312,Z 1478.236,A 0.000,B 0.000,C 90.000,E1 42.405} C_DIS
LIN {X 0.036,Y -224.901,Z 1478.215,A 0.000,B 0.000,C 90.000,E1 38.624} C_DIS
LIN {X -0.094,Y -217.511,Z 1478.193,A 0.000,B 0.000,C 90.000,E1 34.818} C_DIS
LIN {X 0.071,Y -210.952,Z 1478.172,A 0.000,B 0.000,C 90.000,E1 30.875} C_DIS
LIN {X -0.026,Y -205.343,Z 1478.150,A 0.000,B 0.000,C 90.000,E1 26.950} C_DIS
LIN {X -0.025,Y -200.500,Z 1478.127,A 0.000,B 0.000,C 90.000,E1 22.950} C_DIS
LIN {X -0.013,Y -196.321,Z 1478.105,A 0.000,B 0.000,C 90.000,E1 18.906} C_DIS
LIN {X -0.007,Y -192.344,Z 1478.078,A 0.000,B 0.000,C 90.000,E1 14.008} C_DIS
LIN {X 0.080,Y -189.048,Z 1478.046,A 0.000,B 0.000,C 90.000,E1 8.219} C_DIS
LIN {X 0.000,Y -186.694,Z 1478.000,A 0.000,B 0.000,C 90.000,E1 360.000} C_DIS
LIN {X -0.023,Y -186.651,Z 1477.970,A 0.000,B 0.000,C 90.000,E1 354.546} C_DIS
LIN {X 0.057,Y -187.855,Z 1477.937,A 0.000,B 0.000,C 90.000,E1 348.701} C_DIS
LIN {X 0.046,Y -190.534,Z 1477.905,A 0.000,B 0.000,C 90.000,E1 342.906} C_DIS
LIN {X 0.018,Y -194.128,Z 1477.878,A 0.000,B 0.000,C 90.000,E1 337.975} C_DIS
LIN {X 0.003,Y -198.045,Z 1477.855,A 0.000,B 0.000,C 90.000,E1 333.896} C_DIS
LIN {X -0.074,Y -202.999,Z 1477.833,A 0.000,B 0.000,C 90.000,E1 329.871} C_DIS
LIN {X 0.065,Y -207.815,Z 1477.815,A 0.000,B 0.000,C 90.000,E1 326.628} C_DIS
LIN {X -0.080,Y -213.480,Z 1477.797,A 0.000,B 0.000,C 90.000,E1 323.497} C_DIS
LIN {X -0.047,Y -219.973,Z 1477.780,A 0.000,B 0.000,C 90.000,E1 320.356} C_DIS
LIN {X 0.041,Y -228.499,Z 1477.760,A 0.000,B 0.000,C 90.000,E1 316.863} C_DIS
LIN {X -0.078,Y -237.069,Z 1477.744,A 0.000,B 0.000,C 90.000,E1 313.866} C_DIS
LIN {X 0.053,Y -246.567,Z 1477.727,A 0.000,B 0.000,C 90.000,E1 310.862} C_DIS
LIN {X 0.084,Y -256.010,Z 1477.713,A 0.000,B 0.000,C 90.000,E1 308.302} C_DIS
LIN {X 0.000,Y -265.054,Z 1477.701,A 0.000,B 0.000,C 90.000,E1 306.171} C_DIS
LIN {X 0.015,Y -273.344,Z 1477.691,A 0.000,B 0.000,C 90.000,E1 304.405} C_DIS
LIN {X -0.003,Y -282.763,Z 1477.682,A 0.000,B 0.000,C 90.000,E1 302.673} C_DIS
LIN {X 0.058,Y -297.293,Z 1477.668,A 0.000,B 0.000,C 90.000,E1 300.285} C_DIS
LIN {X 0.072,Y -304.143,Z 1477.663,A 0.000,B 0.000,C 90.000,E1 299.283} C_DIS
LIN {X -0.102,Y -314.135,Z 1477.656,A 0.000,B 0.000,C 90.000,E1 298.025} C_DIS
LIN {X 0.084,Y -327.877,Z 1477.647,A 0.000,B 0.000,C 90.000,E1 296.437} C_DIS
LIN {X 0.018,Y -349.564,Z 1477.635,A 0.000,B 0.000,C 90.000,E1 294.207} C_DIS
LIN {X -0.066,Y -360.444,Z 1477.628,A 0.000,B 0.000,C 90.000,E1 293.131} C_DIS
LIN {X 0.075,Y -371.027,Z 1477.622,A 0.000,B 0.000,C 90.000,E1 292.025} C_DIS
LIN {X 0.099,Y -381.523,Z 1477.616,A 0.000,B 0.000,C 90.000,E1 290.918} C_DIS
LIN {X 0.113,Y -391.823,Z 1477.610,A 0.000,B 0.000,C 90.000,E1 289.812} C_DIS
LIN {X -0.126,Y -401.803,Z 1477.604,A 0.000,B 0.000,C 90.000,E1 288.725} C_DIS
LIN {X 0.041,Y -411.240,Z 1477.598,A 0.000,B 0.000,C 90.000,E1 287.583} C_DIS
LIN {X 0.205,Y -417.743,Z 1477.593,A 0.000,B 0.000,C 90.000,E1 286.732} C_DIS
LIN {X -0.092,Y -423.635,Z 1477.589,A 0.000,B 0.000,C 90.000,E1 285.953} C_DIS
LIN {X -0.050,Y -428.858,Z 1477.584,A 0.000,B 0.000,C 90.000,E1 285.134} C_DIS
LIN {X -0.017,Y -431.840,Z 1477.581,A 0.000,B 0.000,C 90.000,E1 284.592} C_DIS
LIN {X 0.114,Y -435.619,Z 1477.577,A 0.000,B 0.000,C 90.000,E1 283.772} C_DIS
LIN {X -0.142,Y -438.668,Z 1477.572,A 0.000,B 0.000,C 90.000,E1 283.008} C_DIS
LIN {X -0.161,Y -440.301,Z 1477.569,A 0.000,B 0.000,C 90.000,E1 282.479} C_DIS
LIN {X -0.168,Y -441.538,Z 1477.566,A 0.000,B 0.000,C 90.000,E1 281.951} C_DIS
LIN {X -0.166,Y -442.339,Z 1477.563,A 0.000,B 0.000,C 90.000,E1 281.422} C_DIS
LIN {X -0.158,Y -442.681,Z 1477.560,A 0.000,B 0.000,C 90.000,E1 280.894} C_DIS
LIN {X -0.147,Y -442.490,Z 1477.557,A 0.000,B 0.000,C 90.000,E1 280.366} C_DIS
LIN {X -0.212,Y -441.752,Z 1477.555,A 0.000,B 0.000,C 90.000,E1 279.849} C_DIS
LIN {X -0.202,Y -440.426,Z 1477.552,A 0.000,B 0.000,C 90.000,E1 279.321} C_DIS
LIN {X 0.165,Y -438.404,Z 1477.549,A 0.000,B 0.000,C 90.000,E1 278.746} C_DIS
LIN {X 0.157,Y -435.618,Z 1477.546,A 0.000,B 0.000,C 90.000,E1 278.219} C_DIS
LIN {X 0.066,Y -431.987,Z 1477.543,A 0.000,B 0.000,C 90.000,E1 277.701} C_DIS
LIN {X -0.040,Y -427.272,Z 1477.540,A 0.000,B 0.000,C 90.000,E1 277.182} C_DIS
LIN {X 0.133,Y -424.470,Z 1477.538,A 0.000,B 0.000,C 90.000,E1 276.891} C_DIS
LIN {X -0.139,Y -418.444,Z 1477.536,A 0.000,B 0.000,C 90.000,E1 276.429} C_DIS
LIN {X 0.075,Y -412.201,Z 1477.533,A 0.000,B 0.000,C 90.000,E1 275.967} C_DIS
LIN {X 0.176,Y -405.808,Z 1477.531,A 0.000,B 0.000,C 90.000,E1 275.568} C_DIS
LIN {X -0.188,Y -399.168,Z 1477.529,A 0.000,B 0.000,C 90.000,E1 275.277} C_DIS
LIN {X -0.108,Y -389.289,Z 1477.527,A 0.000,B 0.000,C 90.000,E1 274.821} C_DIS
LIN {X -0.108,Y -376.503,Z 1477.524,A 0.000,B 0.000,C 90.000,E1 274.302} C_DIS
LIN {X 0.126,Y -361.130,Z 1477.521,A 0.000,B 0.000,C 90.000,E1 273.669} C_DIS
LIN {X -0.144,Y -348.106,Z 1477.518,A 0.000,B 0.000,C 90.000,E1 273.269} C_DIS
LIN {X 0.137,Y -337.837,Z 1477.516,A 0.000,B 0.000,C 90.000,E1 272.922} C_DIS
LIN {X 0.010,Y -327.494,Z 1477.515,A 0.000,B 0.000,C 90.000,E1 272.694} C_DIS
LIN {X 0.065,Y -316.057,Z 1477.514,A 0.000,B 0.000,C 90.000,E1 272.465} C_DIS
LIN {X 0.008,Y -307.790,Z 1477.513,A 0.000,B 0.000,C 90.000,E1 272.350} C_DIS
LIN {X -0.121,Y -299.797,Z 1477.513,A 0.000,B 0.000,C 90.000,E1 272.293} C_DIS
LIN {X -0.107,Y -286.423,Z 1477.512,A 0.000,B 0.000,C 90.000,E1 272.236} C_DIS
LIN {X 0.083,Y -181.229,Z 1477.512,A 0.000,B 0.000,C 90.000,E1 272.178} C_DIS
LIN {X 0.077,Y -181.567,Z 1477.503,A 0.000,B 0.000,C 90.000,E1 270.458} C_DIS
LIN {X 0.066,Y -181.117,Z 1477.489,A 0.000,B 0.000,C 90.000,E1 267.936} C_DIS
LIN {X 0.054,Y -180.906,Z 1477.475,A 0.000,B 0.000,C 90.000,E1 265.412} C_DIS
LIN {X -0.069,Y -180.718,Z 1477.470,A 0.000,B 0.000,C 90.000,E1 264.609} C_DIS
LIN {X 0.029,Y -178.806,Z 1477.442,A 0.000,B 0.000,C 90.000,E1 259.511} C_DIS
LIN {X -0.064,Y -175.850,Z 1477.413,A 0.000,B 0.000,C 90.000,E1 254.448} C_DIS
LIN {X -0.082,Y -173.177,Z 1477.395,A 0.000,B 0.000,C 90.000,E1 251.040} C_DIS
LIN {X 0.080,Y -171.477,Z 1477.380,A 0.000,B 0.000,C 90.000,E1 248.411} C_DIS
LIN {X -0.091,Y -167.707,Z 1477.356,A 0.000,B 0.000,C 90.000,E1 244.152} C_DIS
LIN {X 0.072,Y -166.395,Z 1477.347,A 0.000,B 0.000,C 90.000,E1 242.359} C_DIS
LIN {X 0.064,Y -163.121,Z 1477.327,A 0.000,B 0.000,C 90.000,E1 238.869} C_DIS
LIN {X -0.110,Y -161.072,Z 1477.313,A 0.000,B 0.000,C 90.000,E1 236.294} C_DIS
LIN {X 0.001,Y -157.804,Z 1477.293,A 0.000,B 0.000,C 90.000,E1 232.718} C_DIS
LIN {X -0.061,Y -155.839,Z 1477.278,A 0.000,B 0.000,C 90.000,E1 230.070} C_DIS
LIN {X -0.005,Y -152.090,Z 1477.253,A 0.000,B 0.000,C 90.000,E1 225.567} C_DIS
LIN {X 0.014,Y -150.341,Z 1477.238,A 0.000,B 0.000,C 90.000,E1 222.852} C_DIS
LIN {X 0.035,Y -147.079,Z 1477.213,A 0.000,B 0.000,C 90.000,E1 218.302} C_DIS
LIN {X -0.061,Y -145.652,Z 1477.198,A 0.000,B 0.000,C 90.000,E1 215.598} C_DIS
LIN {X -0.057,Y -143.035,Z 1477.172,A 0.000,B 0.000,C 90.000,E1 211.003} C_DIS
LIN {X 0.069,Y -141.659,Z 1477.152,A 0.000,B 0.000,C 90.000,E1 207.257} C_DIS
LIN {X -0.011,Y -139.447,Z 1477.115,A 0.000,B 0.000,C 90.000,E1 200.791} C_DIS
LIN {X 0.041,Y -139.181,Z 1477.105,A 0.000,B 0.000,C 90.000,E1 198.906} C_DIS
LIN {X -0.067,Y -138.320,Z 1477.053,A 0.000,B 0.000,C 90.000,E1 189.613} C_DIS
LIN {X -0.060,Y -139.464,Z 1477.007,A 0.000,B 0.000,C 90.000,E1 181.203} C_DIS
LIN {X 0.019,Y -141.027,Z 1476.975,A 0.000,B 0.000,C 90.000,E1 175.584} C_DIS
LIN {X -0.025,Y -142.393,Z 1476.960,A 0.000,B 0.000,C 90.000,E1 172.818} C_DIS
LIN {X 0.037,Y -144.625,Z 1476.934,A 0.000,B 0.000,C 90.000,E1 168.173} C_DIS
LIN {X -0.044,Y -147.820,Z 1476.909,A 0.000,B 0.000,C 90.000,E1 163.614} C_DIS
LIN {X 0.043,Y -150.511,Z 1476.889,A 0.000,B 0.000,C 90.000,E1 159.934} C_DIS
LIN {X -0.078,Y -153.971,Z 1476.869,A 0.000,B 0.000,C 90.000,E1 156.357} C_DIS
LIN {X -0.016,Y -157.383,Z 1476.849,A 0.000,B 0.000,C 90.000,E1 152.743} C_DIS
LIN {X -0.074,Y -161.586,Z 1476.829,A 0.000,B 0.000,C 90.000,E1 149.203} C_DIS
LIN {X -0.063,Y -165.783,Z 1476.809,A 0.000,B 0.000,C 90.000,E1 145.674} C_DIS
LIN {X -0.077,Y -170.744,Z 1476.790,A 0.000,B 0.000,C 90.000,E1 142.190} C_DIS
LIN {X 0.080,Y -175.616,Z 1476.771,A 0.000,B 0.000,C 90.000,E1 138.690} C_DIS
LIN {X -0.050,Y -181.233,Z 1476.752,A 0.000,B 0.000,C 90.000,E1 135.324} C_DIS
LIN {X 0.081,Y -186.701,Z 1476.733,A 0.000,B 0.000,C 90.000,E1 131.919} C_DIS
LIN {X 0.033,Y -191.301,Z 1476.719,A 0.000,B 0.000,C 90.000,E1 129.439} C_DIS
LIN {X -0.036,Y -197.129,Z 1476.701,A 0.000,B 0.000,C 90.000,E1 126.171} C_DIS
LIN {X -0.015,Y -201.164,Z 1476.690,A 0.000,B 0.000,C 90.000,E1 124.119} C_DIS
LIN {X 0.036,Y -201.220,Z 1476.689,A 0.000,B 0.000,C 90.000,E1 124.072} C_DIS
LIN {X -0.004,Y -313.325,Z 1476.689,A 0.000,B 0.000,C 90.000,E1 124.072} C_DIS
LIN {X -0.089,Y -319.267,Z 1476.688,A 0.000,B 0.000,C 90.000,E1 123.913} C_DIS
LIN {X 0.092,Y -321.741,Z 1476.687,A 0.000,B 0.000,C 90.000,E1 123.706} C_DIS
LIN {X 0.058,Y -325.570,Z 1476.685,A 0.000,B 0.000,C 90.000,E1 123.293} C_DIS
LIN {X -0.010,Y -327.457,Z 1476.683,A 0.000,B 0.000,C 90.000,E1 123.007} C_DIS
LIN {X 0.017,Y -328.935,Z 1476.682,A 0.000,B 0.000,C 90.000,E1 122.704} C_DIS
LIN {X 0.092,Y -343.626,Z 1476.661,A 0.000,B 0.000,C 90.000,E1 118.949} C_DIS
LIN {X -0.076,Y -356.170,Z 1476.646,A 0.000,B 0.000,C 90.000,E1 116.232} C_DIS
LIN {X 0.115,Y -370.219,Z 1476.631,A 0.000,B 0.000,C 90.000,E1 113.515} C_DIS
LIN {X -0.207,Y -384.064,Z 1476.618,A 0.000,B 0.000,C 90.000,E1 111.227} C_DIS
LIN {X 0.034,Y -399.287,Z 1476.605,A 0.000,B 0.000,C 90.000,E1 108.906} C_DIS
LIN {X 0.020,Y -415.994,Z 1476.593,A 0.000,B 0.000,C 90.000,E1 106.677} C_DIS
LIN {X 0.188,Y -434.303,Z 1476.581,A 0.000,B 0.000,C 90.000,E1 104.481} C_DIS
LIN {X 0.081,Y -454.033,Z 1476.569,A 0.000,B 0.000,C 90.000,E1 102.411} C_DIS
LIN {X 0.102,Y -474.383,Z 1476.558,A 0.000,B 0.000,C 90.000,E1 100.489} C_DIS
LIN {X 0.042,Y -487.347,Z 1476.552,A 0.000,B 0.000,C 90.000,E1 99.378} C_DIS
LIN {X 0.110,Y -489.765,Z 1476.551,A 0.000,B 0.000,C 90.000,E1 99.151} C_DIS
LIN {X 0.166,Y -491.672,Z 1476.550,A 0.000,B 0.000,C 90.000,E1 98.916} C_DIS
LIN {X 0.148,Y -493.125,Z 1476.548,A 0.000,B 0.000,C 90.000,E1 98.690} C_DIS
LIN {X -0.037,Y -495.152,Z 1476.546,A 0.000,B 0.000,C 90.000,E1 98.219} C_DIS
LIN {X 0.204,Y -496.021,Z 1476.543,A 0.000,B 0.000,C 90.000,E1 97.701} C_DIS
LIN {X -0.033,Y -495.884,Z 1476.540,A 0.000,B 0.000,C 90.000,E1 97.239} C_DIS
LIN {X 0.227,Y -494.726,Z 1476.537,A 0.000,B 0.000,C 90.000,E1 96.720} C_DIS
LIN {X 0.138,Y -493.709,Z 1476.536,A 0.000,B 0.000,C 90.000,E1 96.486} C_DIS
LIN {X -0.006,Y -492.334,Z 1476.535,A 0.000,B 0.000,C 90.000,E1 96.258} C_DIS
LIN {X 0.179,Y -482.346,Z 1476.527,A 0.000,B 0.000,C 90.000,E1 94.759} C_DIS
LIN {X -0.041,Y -471.736,Z 1476.517,A 0.000,B 0.000,C 90.000,E1 93.037} C_DIS
LIN {X -0.062,Y -463.736,Z 1476.510,A 0.000,B 0.000,C 90.000,E1 91.776} C_DIS
LIN {X 0.023,Y -453.607,Z 1476.501,A 0.000,B 0.000,C 90.000,E1 90.229} C_DIS
LIN {X -0.123,Y -439.800,Z 1476.490,A 0.000,B 0.000,C 90.000,E1 88.165} C_DIS
LIN {X 0.143,Y -427.757,Z 1476.479,A 0.000,B 0.000,C 90.000,E1 86.274} C_DIS
LIN {X 0.210,Y -415.671,Z 1476.469,A 0.000,B 0.000,C 90.000,E1 84.375} C_DIS
LIN {X -0.028,Y -405.247,Z 1476.460,A 0.000,B 0.000,C 90.000,E1 82.761} C_DIS
LIN {X 0.074,Y -392.950,Z 1476.449,A 0.000,B 0.000,C 90.000,E1 80.792} C_DIS
LIN {X 0.062,Y -375.907,Z 1476.433,A 0.000,B 0.000,C 90.000,E1 77.937} C_DIS
LIN {X 0.111,Y -362.775,Z 1476.420,A 0.000,B 0.000,C 90.000,E1 75.589} C_DIS
LIN {X 0.088,Y -351.484,Z 1476.408,A 0.000,B 0.000,C 90.000,E1 73.504} C_DIS
LIN {X -0.063,Y -338.624,Z 1476.395,A 0.000,B 0.000,C 90.000,E1 71.094} C_DIS
LIN {X -0.021,Y -324.336,Z 1476.379,A 0.000,B 0.000,C 90.000,E1 68.284} C_DIS
LIN {X -0.167,Y -307.990,Z 1476.360,A 0.000,B 0.000,C 90.000,E1 64.793} C_DIS
LIN {X 0.066,Y -294.275,Z 1476.342,A 0.000,B 0.000,C 90.000,E1 61.463} C_DIS
LIN {X -0.040,Y -282.759,Z 1476.325,A 0.000,B 0.000,C 90.000,E1 58.456} C_DIS
LIN {X -0.086,Y -272.968,Z 1476.309,A 0.000,B 0.000,C 90.000,E1 55.722} C_DIS
LIN {X -0.007,Y -262.277,Z 1476.292,A 0.000,B 0.000,C 90.000,E1 52.557} C_DIS
LIN {X 0.023,Y -251.030,Z 1476.272,A 0.000,B 0.000,C 90.000,E1 48.976} C_DIS
LIN {X 0.051,Y -240.758,Z 1476.252,A 0.000,B 0.000,C 90.000,E1 45.324} C_DIS
LIN {X 0.088,Y -231.587,Z 1476.231,A 0.000,B 0.000,C 90.000,E1 41.595} C_DIS
LIN {X 0.077,Y -223.413,Z 1476.210,A 0.000,B 0.000,C 90.000,E1 37.810} C_DIS
LIN {X -0.053,Y -216.277,Z 1476.189,A 0.000,B 0.000,C 90.000,E1 33.992} C_DIS
LIN {X -0.035,Y -209.946,Z 1476.167,A 0.000,B 0.000,C 90.000,E1 30.079} C_DIS
LIN {X 0.018,Y -204.523,Z 1476.145,A 0.000,B 0.000,C 90.000,E1 26.104} C_DIS
LIN {X 0.086,Y -199.804,Z 1476.123,A 0.000,B 0.000,C 90.000,E1 22.078} C_DIS
LIN {X 0.005,Y -195.798,Z 1476.100,A 0.000,B 0.000,C 90.000,E1 18.055} C_DIS
LIN {X -0.067,Y -192.017,Z 1476.073,A 0.000,B 0.000,C 90.000,E1 13.175} C_DIS
LIN {X -0.068,Y -188.921,Z 1476.041,A 0.000,B 0.000,C 90.000,E1 7.409} C_DIS
LIN {X -0.034,Y -186.921,Z 1475.997,A 0.000,B 0.000,C 90.000,E1 359.542} C_DIS
LIN {X 0.083,Y -186.997,Z 1475.965,A 0.000,B 0.000,C 90.000,E1 353.685} C_DIS
LIN {X 0.016,Y -188.686,Z 1475.928,A 0.000,B 0.000,C 90.000,E1 347.061} C_DIS
LIN {X 0.014,Y -191.792,Z 1475.896,A 0.000,B 0.000,C 90.000,E1 341.275} C_DIS
LIN {X -0.008,Y -195.742,Z 1475.869,A 0.000,B 0.000,C 90.000,E1 336.357} C_DIS
LIN {X 0.019,Y -200.073,Z 1475.846,A 0.000,B 0.000,C 90.000,E1 332.281} C_DIS
LIN {X 0.033,Y -205.422,Z 1475.824,A 0.000,B 0.000,C 90.000,E1 328.250} C_DIS
LIN {X 0.061,Y -210.700,Z 1475.806,A 0.000,B 0.000,C 90.000,E1 325.055} C_DIS
LIN {X 0.064,Y -216.740,Z 1475.788,A 0.000,B 0.000,C 90.000,E1 321.904} C_DIS
LIN {X 0.011,Y -223.797,Z 1475.771,A 0.000,B 0.000,C 90.000,E1 318.809} C_DIS
LIN {X 0.084,Y -231.746,Z 1475.754,A 0.000,B 0.000,C 90.000,E1 315.729} C_DIS
LIN {X 0.030,Y -241.824,Z 1475.735,A 0.000,B 0.000,C 90.000,E1 312.366} C_DIS
LIN {X -0.048,Y -250.631,Z 1475.721,A 0.000,B 0.000,C 90.000,E1 309.806} C_DIS
LIN {X 0.119,Y -260.575,Z 1475.707,A 0.000,B 0.000,C 90.000,E1 307.237} C_DIS
LIN {X 0.128,Y -270.044,Z 1475.695,A 0.000,B 0.000,C 90.000,E1 305.105} C_DIS
LIN {X 0.130,Y -277.068,Z 1475.687,A 0.000,B 0.000,C 90.000,E1 303.706} C_DIS
LIN {X -0.040,Y -290.957,Z 1475.674,A 0.000,B 0.000,C 90.000,E1 301.337} C_DIS
LIN {X -0.087,Y -299.534,Z 1475.667,A 0.000,B 0.000,C 90.000,E1 300.001} C_DIS
LIN {X -0.052,Y -306.580,Z 1475.661,A 0.000,B 0.000,C 90.000,E1 298.999} C_DIS
LIN {X -0.070,Y -314.235,Z 1475.656,A 0.000,B 0.000,C 90.000,E1 298.025} C_DIS
LIN {X -0.021,Y -327.260,Z 1475.647,A 0.000,B 0.000,C 90.000,E1 296.539} C_DIS
LIN {X 0.077,Y -349.125,Z 1475.635,A 0.000,B 0.000,C 90.000,E1 294.259} C_DIS
LIN {X -0.139,Y -360.001,Z 1475.629,A 0.000,B 0.000,C 90.000,E1 293.206} C_DIS
LIN {X 0.062,Y -370.731,Z 1475.623,A 0.000,B 0.000,C 90.000,E1 292.078} C_DIS
LIN {X 0.128,Y -381.163,Z 1475.617,A 0.000,B 0.000,C 90.000,E1 290.972} C_DIS
LIN {X 0.015,Y -391.463,Z 1475.610,A 0.000,B 0.000,C 90.000,E1 289.885} C_DIS
LIN {X -0.096,Y -401.449,Z 1475.604,A 0.000,B 0.000,C 90.000,E1 288.779} C_DIS
LIN {X 0.083,Y -410.962,Z 1475.598,A 0.000,B 0.000,C 90.000,E1 287.638} C_DIS
LIN {X 0.122,Y -417.516,Z 1475.594,A 0.000,B 0.000,C 90.000,E1 286.804} C_DIS
LIN {X -0.174,Y -423.500,Z 1475.589,A 0.000,B 0.000,C 90.000,E1 286.024} C_DIS
LIN {X -0.018,Y -428.769,Z 1475.584,A 0.000,B 0.000,C 90.000,E1 285.190} C_DIS
LIN {X -0.096,Y -431.813,Z 1475.581,A 0.000,B 0.000,C 90.000,E1 284.662} C_DIS
LIN {X 0.143,Y -435.677,Z 1475.577,A 0.000,B 0.000,C 90.000,E1 283.828} C_DIS
LIN {X -0.115,Y -438.777,Z 1475.573,A 0.000,B 0.000,C 90.000,E1 283.063} C_DIS
LIN {X -0.133,Y -440.465,Z 1475.570,A 0.000,B 0.000,C 90.000,E1 282.535} C_DIS
LIN {X -0.140,Y -441.744,Z 1475.567,A 0.000,B 0.000,C 90.000,E1 282.007} C_DIS
LIN {X -0.137,Y -442.602,Z 1475.564,A 0.000,B 0.000,C 90.000,E1 281.478} C_DIS
LIN {X -0.130,Y -443.038,Z 1475.561,A 0.000,B 0.000,C 90.000,E1 280.950} C_DIS
LIN {X -0.117,Y -442.935,Z 1475.558,A 0.000,B 0.000,C 90.000,E1 280.423} C_DIS
LIN {X -0.182,Y -442.322,Z 1475.555,A 0.000,B 0.000,C 90.000,E1 279.905} C_DIS
LIN {X -0.169,Y -441.078,Z 1475.552,A 0.000,B 0.000,C 90.000,E1 279.378} C_DIS
LIN {X 0.201,Y -439.194,Z 1475.549,A 0.000,B 0.000,C 90.000,E1 278.803} C_DIS
LIN {X 0.196,Y -436.530,Z 1475.546,A 0.000,B 0.000,C 90.000,E1 278.276} C_DIS
LIN {X 0.109,Y -433.047,Z 1475.543,A 0.000,B 0.000,C 90.000,E1 277.757} C_DIS
LIN {X 0.008,Y -428.530,Z 1475.540,A 0.000,B 0.000,C 90.000,E1 277.239} C_DIS
LIN {X -0.114,Y -422.798,Z 1475.537,A 0.000,B 0.000,C 90.000,E1 276.720} C_DIS
LIN {X -0.204,Y -416.664,Z 1475.535,A 0.000,B 0.000,C 90.000,E1 276.258} C_DIS
LIN {X 0.141,Y -410.357,Z 1475.532,A 0.000,B 0.000,C 90.000,E1 275.796} C_DIS
LIN {X -0.057,Y -403.848,Z 1475.530,A 0.000,B 0.000,C 90.000,E1 275.454} C_DIS
LIN {X -0.120,Y -394.053,Z 1475.528,A 0.000,B 0.000,C 90.000,E1 274.992} C_DIS
LIN {X 0.162,Y -381.244,Z 1475.525,A 0.000,B 0.000,C 90.000,E1 274.416} C_DIS
LIN {X -0.089,Y -362.480,Z 1475.521,A 0.000,B 0.000,C 90.000,E1 273.726} C_DIS
LIN {X -0.027,Y -349.396,Z 1475.518,A 0.000,B 0.000,C 90.000,E1 273.269} C_DIS
LIN {X -0.110,Y -339.195,Z 1475.516,A 0.000,B 0.000,C 90.000,E1 272.980} C_DIS
LIN {X -0.028,Y -325.279,Z 1475.515,A 0.000,B 0.000,C 90.000,E1 272.636} C_DIS
LIN {X 0.116,Y -313.663,Z 1475.514,A 0.000,B 0.000,C 90.000,E1 272.407} C_DIS
LIN {X 0.103,Y -304.819,Z 1475.513,A 0.000,B 0.000,C 90.000,E1 272.293} C_DIS
LIN {X -0.053,Y -292.015,Z 1475.512,A 0.000,B 0.000,C 90.000,E1 272.236} C_DIS
LIN {X -0.067,Y -181.228,Z 1475.512,A 0.000,B 0.000,C 90.000,E1 272.236} C_DIS
LIN {X -0.088,Y -181.567,Z 1475.503,A 0.000,B 0.000,C 90.000,E1 270.516} C_DIS
LIN {X 0.083,Y -181.119,Z 1475.489,A 0.000,B 0.000,C 90.000,E1 267.936} C_DIS
LIN {X 0.071,Y -180.907,Z 1475.475,A 0.000,B 0.000,C 90.000,E1 265.412} C_DIS
LIN {X -0.053,Y -180.720,Z 1475.470,A 0.000,B 0.000,C 90.000,E1 264.609} C_DIS
LIN {X 0.046,Y -178.809,Z 1475.442,A 0.000,B 0.000,C 90.000,E1 259.511} C_DIS
LIN {X -0.048,Y -175.854,Z 1475.414,A 0.000,B 0.000,C 90.000,E1 254.448} C_DIS
LIN {X -0.065,Y -173.180,Z 1475.395,A 0.000,B 0.000,C 90.000,E1 251.040} C_DIS
LIN {X -0.063,Y -171.481,Z 1475.380,A 0.000,B 0.000,C 90.000,E1 248.465} C_DIS
LIN {X -0.075,Y -167.711,Z 1475.356,A 0.000,B 0.000,C 90.000,E1 244.152} C_DIS
LIN {X -0.059,Y -166.401,Z 1475.347,A 0.000,B 0.000,C 90.000,E1 242.410} C_DIS
LIN {X 0.079,Y -163.126,Z 1475.327,A 0.000,B 0.000,C 90.000,E1 238.869} C_DIS
LIN {X -0.094,Y -161.077,Z 1475.313,A 0.000,B 0.000,C 90.000,E1 236.294} C_DIS
LIN {X 0.017,Y -157.808,Z 1475.293,A 0.000,B 0.000,C 90.000,E1 232.718} C_DIS
LIN {X -0.045,Y -155.844,Z 1475.278,A 0.000,B 0.000,C 90.000,E1 230.070} C_DIS
LIN {X 0.011,Y -152.094,Z 1475.253,A 0.000,B 0.000,C 90.000,E1 225.567} C_DIS
LIN {X 0.030,Y -150.344,Z 1475.238,A 0.000,B 0.000,C 90.000,E1 222.852} C_DIS
LIN {X 0.051,Y -147.082,Z 1475.213,A 0.000,B 0.000,C 90.000,E1 218.302} C_DIS
LIN {X -0.046,Y -145.655,Z 1475.198,A 0.000,B 0.000,C 90.000,E1 215.598} C_DIS
LIN {X -0.042,Y -143.038,Z 1475.172,A 0.000,B 0.000,C 90.000,E1 211.003} C_DIS
LIN {X -0.042,Y -141.661,Z 1475.152,A 0.000,B 0.000,C 90.000,E1 207.308} C_DIS
LIN {X 0.003,Y -139.449,Z 1475.115,A 0.000,B 0.000,C 90.000,E1 200.791} C_DIS
LIN {X 0.056,Y -139.182,Z 1475.105,A 0.000,B 0.000,C 90.000,E1 198.906} C_DIS
LIN {X -0.052,Y -138.321,Z 1475.053,A 0.000,B 0.000,C 90.000,E1 189.613} C_DIS
LIN {X -0.046,Y -139.464,Z 1475.007,A 0.000,B 0.000,C 90.000,E1 181.203} C_DIS
LIN {X 0.034,Y -141.025,Z 1474.976,A 0.000,B 0.000,C 90.000,E1 175.584} C_DIS
LIN {X -0.011,Y -142.390,Z 1474.960,A 0.000,B 0.000,C 90.000,E1 172.818} C_DIS
LIN {X 0.052,Y -144.621,Z 1474.934,A 0.000,B 0.000,C 90.000,E1 168.173} C_DIS
LIN {X -0.029,Y -147.816,Z 1474.909,A 0.000,B 0.000,C 90.000,E1 163.614} C_DIS
LIN {X 0.058,Y -150.505,Z 1474.889,A 0.000,B 0.000,C 90.000,E1 159.934} C_DIS
LIN {X -0.063,Y -153.965,Z 1474.869,A 0.000,B 0.000,C 90.000,E1 156.357} C_DIS
LIN {X 0.000,Y -157.377,Z 1474.849,A 0.000,B 0.000,C 90.000,E1 152.743} C_DIS
LIN {X -0.058,Y -161.579,Z 1474.829,A 0.000,B 0.000,C 90.000,E1 149.203} C_DIS
LIN {X -0.047,Y -165.776,Z 1474.809,A 0.000,B 0.000,C 90.000,E1 145.674} C_DIS
LIN {X -0.061,Y -170.735,Z 1474.790,A 0.000,B 0.000,C 90.000,E1 142.190} C_DIS
LIN {X -0.018,Y -175.608,Z 1474.771,A 0.000,B 0.000,C 90.000,E1 138.728} C_DIS
LIN {X -0.033,Y -181.224,Z 1474.752,A 0.000,B 0.000,C 90.000,E1 135.324} C_DIS
LIN {X 0.099,Y -186.691,Z 1474.733,A 0.000,B 0.000,C 90.000,E1 131.919} C_DIS
LIN {X 0.051,Y -191.292,Z 1474.719,A 0.000,B 0.000,C 90.000,E1 129.439} C_DIS
LIN {X -0.018,Y -197.120,Z 1474.701,A 0.000,B 0.000,C 90.000,E1 126.171} C_DIS
LIN {X -0.035,Y -201.174,Z 1474.689,A 0.000,B 0.000,C 90.000,E1 124.119} C_DIS
LIN {X -0.114,Y -313.100,Z 1474.689,A 0.000,B 0.000,C 90.000,E1 124.119} C_DIS
LIN {X 0.026,Y -315.165,Z 1474.689,A 0.000,B 0.000,C 90.000,E1 124.072} C_DIS
LIN {X -0.059,Y -319.515,Z 1474.688,A 0.000,B 0.000,C 90.000,E1 123.913} C_DIS
LIN {X 0.122,Y -321.877,Z 1474.687,A 0.000,B 0.000,C 90.000,E1 123.706} C_DIS
LIN {X -0.011,Y -325.728,Z 1474.685,A 0.000,B 0.000,C 90.000,E1 123.293} C_DIS
LIN {X 0.152,Y -327.592,Z 1474.683,A 0.000,B 0.000,C 90.000,E1 122.959} C_DIS
LIN {X 0.039,Y -329.050,Z 1474.682,A 0.000,B 0.000,C 90.000,E1 122.673} C_DIS
LIN {X -0.052,Y -342.408,Z 1474.662,A 0.000,B 0.000,C 90.000,E1 119.255} C_DIS
LIN {X 0.044,Y -354.809,Z 1474.647,A 0.000,B 0.000,C 90.000,E1 116.488} C_DIS
LIN {X -0.131,Y -368.697,Z 1474.632,A 0.000,B 0.000,C 90.000,E1 113.823} C_DIS
LIN {X -0.006,Y -382.390,Z 1474.619,A 0.000,B 0.000,C 90.000,E1 111.461} C_DIS
LIN {X 0.193,Y -397.450,Z 1474.606,A 0.000,B 0.000,C 90.000,E1 109.141} C_DIS
LIN {X 0.136,Y -413.982,Z 1474.594,A 0.000,B 0.000,C 90.000,E1 106.913} C_DIS
LIN {X -0.162,Y -432.100,Z 1474.582,A 0.000,B 0.000,C 90.000,E1 104.773} C_DIS
LIN {X 0.037,Y -451.708,Z 1474.570,A 0.000,B 0.000,C 90.000,E1 102.647} C_DIS
LIN {X -0.011,Y -471.996,Z 1474.560,A 0.000,B 0.000,C 90.000,E1 100.715} C_DIS
LIN {X -0.124,Y -487.550,Z 1474.552,A 0.000,B 0.000,C 90.000,E1 99.378} C_DIS
LIN {X -0.056,Y -489.899,Z 1474.551,A 0.000,B 0.000,C 90.000,E1 99.151} C_DIS
LIN {X -0.035,Y -491.774,Z 1474.550,A 0.000,B 0.000,C 90.000,E1 98.916} C_DIS
LIN {X -0.016,Y -493.197,Z 1474.548,A 0.000,B 0.000,C 90.000,E1 98.681} C_DIS
LIN {X 0.216,Y -495.133,Z 1474.546,A 0.000,B 0.000,C 90.000,E1 98.163} C_DIS
LIN {X -0.032,Y -495.928,Z 1474.543,A 0.000,B 0.000,C 90.000,E1 97.701} C_DIS
LIN {X 0.222,Y -495.724,Z 1474.540,A 0.000,B 0.000,C 90.000,E1 97.182} C_DIS
LIN {X -0.010,Y -494.491,Z 1474.537,A 0.000,B 0.000,C 90.000,E1 96.720} C_DIS
LIN {X -0.099,Y -493.428,Z 1474.536,A 0.000,B 0.000,C 90.000,E1 96.486} C_DIS
LIN {X -0.242,Y -491.996,Z 1474.535,A 0.000,B 0.000,C 90.000,E1 96.258} C_DIS
LIN {X -0.059,Y -482.012,Z 1474.526,A 0.000,B 0.000,C 90.000,E1 94.759} C_DIS
LIN {X 0.003,Y -469.847,Z 1474.515,A 0.000,B 0.000,C 90.000,E1 92.751} C_DIS
LIN {X -0.048,Y -461.706,Z 1474.508,A 0.000,B 0.000,C 90.000,E1 91.489} C_DIS
LIN {X 0.002,Y -451.497,Z 1474.500,A 0.000,B 0.000,C 90.000,E1 89.943} C_DIS
LIN {X -0.189,Y -437.761,Z 1474.488,A 0.000,B 0.000,C 90.000,E1 87.879} C_DIS
LIN {X 0.037,Y -425.764,Z 1474.478,A 0.000,B 0.000,C 90.000,E1 85.988} C_DIS
LIN {X 0.056,Y -413.678,Z 1474.467,A 0.000,B 0.000,C 90.000,E1 84.090} C_DIS
LIN {X -0.166,Y -403.287,Z 1474.458,A 0.000,B 0.000,C 90.000,E1 82.470} C_DIS
LIN {X -0.091,Y -391.033,Z 1474.447,A 0.000,B 0.000,C 90.000,E1 80.500} C_DIS
LIN {X -0.152,Y -374.111,Z 1474.431,A 0.000,B 0.000,C 90.000,E1 77.645} C_DIS
LIN {X -0.049,Y -361.031,Z 1474.418,A 0.000,B 0.000,C 90.000,E1 75.283} C_DIS
LIN {X -0.100,Y -349.729,Z 1474.407,A 0.000,B 0.000,C 90.000,E1 73.196} C_DIS
LIN {X 0.041,Y -338.465,Z 1474.395,A 0.000,B 0.000,C 90.000,E1 71.040} C_DIS
LIN {X 0.068,Y -324.193,Z 1474.379,A 0.000,B 0.000,C 90.000,E1 68.230} C_DIS
LIN {X 0.037,Y -307.847,Z 1474.360,A 0.000,B 0.000,C 90.000,E1 64.717} C_DIS
LIN {X 0.006,Y -294.127,Z 1474.341,A 0.000,B 0.000,C 90.000,E1 61.435} C_DIS
LIN {X 0.004,Y -282.610,Z 1474.324,A 0.000,B 0.000,C 90.000,E1 58.408} C_DIS
LIN {X -0.054,Y -272.848,Z 1474.309,A 0.000,B 0.000,C 90.000,E1 55.674} C_DIS
LIN {X 0.011,Y -262.189,Z 1474.292,A 0.000,B 0.000,C 90.000,E1 52.512} C_DIS
LIN {X 0.029,Y -250.992,Z 1474.272,A 0.000,B 0.000,C 90.000,E1 48.933} C_DIS
LIN {X -0.125,Y -240.761,Z 1474.252,A 0.000,B 0.000,C 90.000,E1 45.324} C_DIS
LIN {X -0.081,Y -231.620,Z 1474.231,A 0.000,B 0.000,C 90.000,E1 41.595} C_DIS
LIN {X -0.085,Y -223.513,Z 1474.210,A 0.000,B 0.000,C 90.000,E1 37.810} C_DIS
LIN {X 0.094,Y -216.430,Z 1474.189,A 0.000,B 0.000,C 90.000,E1 33.913} C_DIS
LIN {X 0.107,Y -210.116,Z 1474.167,A 0.000,B 0.000,C 90.000,E1 30.001} C_DIS
LIN {X 0.066,Y -204.708,Z 1474.145,A 0.000,B 0.000,C 90.000,E1 26.052} C_DIS
LIN {X -0.041,Y -200.011,Z 1474.123,A 0.000,B 0.000,C 90.000,E1 22.078} C_DIS
LIN {X -0.042,Y -195.320,Z 1474.096,A 0.000,B 0.000,C 90.000,E1 17.221} C_DIS
LIN {X 0.012,Y -191.710,Z 1474.068,A 0.000,B 0.000,C 90.000,E1 12.299} C_DIS
LIN {X -0.031,Y -188.835,Z 1474.036,A 0.000,B 0.000,C 90.000,E1 6.543} C_DIS
LIN {X -0.034,Y -187.179,Z 1473.997,A 0.000,B 0.000,C 90.000,E1 359.542} C_DIS
LIN {X -0.092,Y -187.261,Z 1473.965,A 0.000,B 0.000,C 90.000,E1 353.742} C_DIS
LIN {X 0.039,Y -188.917,Z 1473.928,A 0.000,B 0.000,C 90.000,E1 347.061} C_DIS
LIN {X 0.048,Y -191.993,Z 1473.896,A 0.000,B 0.000,C 90.000,E1 341.275} C_DIS
LIN {X 0.034,Y -195.904,Z 1473.869,A 0.000,B 0.000,C 90.000,E1 336.357} C_DIS
LIN {X 0.066,Y -200.204,Z 1473.846,A 0.000,B 0.000,C 90.000,E1 332.281} C_DIS
LIN {X -0.023,Y -205.551,Z 1473.824,A 0.000,B 0.000,C 90.000,E1 328.280} C_DIS
LIN {X -0.054,Y -210.829,Z 1473.806,A 0.000,B 0.000,C 90.000,E1 325.102} C_DIS
LIN {X 0.127,Y -216.878,Z 1473.789,A 0.000,B 0.000,C 90.000,E1 321.904} C_DIS
LIN {X -0.090,Y -223.944,Z 1473.771,A 0.000,B 0.000,C 90.000,E1 318.852} C_DIS
LIN {X -0.004,Y -231.891,Z 1473.754,A 0.000,B 0.000,C 90.000,E1 315.769} C_DIS
LIN {X 0.112,Y -241.976,Z 1473.735,A 0.000,B 0.000,C 90.000,E1 312.366} C_DIS
LIN {X 0.040,Y -250.793,Z 1473.721,A 0.000,B 0.000,C 90.000,E1 309.806} C_DIS
LIN {X -0.112,Y -262.242,Z 1473.705,A 0.000,B 0.000,C 90.000,E1 306.950} C_DIS
LIN {X -0.079,Y -271.854,Z 1473.693,A 0.000,B 0.000,C 90.000,E1 304.818} C_DIS
LIN {X -0.061,Y -279.084,Z 1473.686,A 0.000,B 0.000,C 90.000,E1 303.420} C_DIS
LIN {X 0.058,Y -293.105,Z 1473.672,A 0.000,B 0.000,C 90.000,E1 301.003} C_DIS
LIN {X 0.039,Y -301.846,Z 1473.665,A 0.000,B 0.000,C 90.000,E1 299.667} C_DIS
LIN {X -0.057,Y -309.076,Z 1473.659,A 0.000,B 0.000,C 90.000,E1 298.693} C_DIS
LIN {X -0.089,Y -319.429,Z 1473.652,A 0.000,B 0.000,C 90.000,E1 297.436} C_DIS
LIN {X -0.166,Y -340.790,Z 1473.640,A 0.000,B 0.000,C 90.000,E1 295.155} C_DIS
LIN {X -0.068,Y -354.471,Z 1473.632,A 0.000,B 0.000,C 90.000,E1 293.770} C_DIS
LIN {X 0.051,Y -367.946,Z 1473.624,A 0.000,B 0.000,C 90.000,E1 292.386} C_DIS
LIN {X 0.109,Y -378.495,Z 1473.618,A 0.000,B 0.000,C 90.000,E1 291.280} C_DIS
LIN {X -0.196,Y -391.434,Z 1473.611,A 0.000,B 0.000,C 90.000,E1 289.939} C_DIS
LIN {X 0.092,Y -403.907,Z 1473.603,A 0.000,B 0.000,C 90.000,E1 288.489} C_DIS
LIN {X -0.101,Y -413.290,Z 1473.597,A 0.000,B 0.000,C 90.000,E1 287.402} C_DIS
LIN {X 0.085,Y -419.710,Z 1473.592,A 0.000,B 0.000,C 90.000,E1 286.551} C_DIS
LIN {X 0.089,Y -425.501,Z 1473.588,A 0.000,B 0.000,C 90.000,E1 285.733} C_DIS
LIN {X -0.141,Y -430.540,Z 1473.583,A 0.000,B 0.000,C 90.000,E1 284.954} C_DIS
LIN {X 0.081,Y -434.675,Z 1473.578,A 0.000,B 0.000,C 90.000,E1 284.120} C_DIS
LIN {X 0.041,Y -437.013,Z 1473.576,A 0.000,B 0.000,C 90.000,E1 283.592} C_DIS
LIN {X 0.017,Y -439.042,Z 1473.573,A 0.000,B 0.000,C 90.000,E1 283.063} C_DIS
LIN {X 0.000,Y -440.743,Z 1473.570,A 0.000,B 0.000,C 90.000,E1 282.535} C_DIS
LIN {X -0.005,Y -442.031,Z 1473.567,A 0.000,B 0.000,C 90.000,E1 282.007} C_DIS
LIN {X -0.001,Y -442.970,Z 1473.564,A 0.000,B 0.000,C 90.000,E1 281.478} C_DIS
LIN {X 0.010,Y -443.406,Z 1473.561,A 0.000,B 0.000,C 90.000,E1 280.950} C_DIS
LIN {X -0.057,Y -443.335,Z 1473.558,A 0.000,B 0.000,C 90.000,E1 280.433} C_DIS
LIN {X -0.039,Y -442.773,Z 1473.555,A 0.000,B 0.000,C 90.000,E1 279.905} C_DIS
LIN {X -0.025,Y -441.531,Z 1473.552,A 0.000,B 0.000,C 90.000,E1 279.378} C_DIS
LIN {X -0.086,Y -439.763,Z 1473.549,A 0.000,B 0.000,C 90.000,E1 278.859} C_DIS
LIN {X -0.151,Y -437.152,Z 1473.546,A 0.000,B 0.000,C 90.000,E1 278.341} C_DIS
LIN {X 0.056,Y -435.601,Z 1473.545,A 0.000,B 0.000,C 90.000,E1 278.049} C_DIS
LIN {X -0.032,Y -431.720,Z 1473.542,A 0.000,B 0.000,C 90.000,E1 277.530} C_DIS
LIN {X 0.161,Y -429.354,Z 1473.540,A 0.000,B 0.000,C 90.000,E1 277.239} C_DIS
LIN {X 0.043,Y -423.763,Z 1473.537,A 0.000,B 0.000,C 90.000,E1 276.720} C_DIS
LIN {X -0.139,Y -417.456,Z 1473.535,A 0.000,B 0.000,C 90.000,E1 276.258} C_DIS
LIN {X -0.197,Y -411.241,Z 1473.532,A 0.000,B 0.000,C 90.000,E1 275.853} C_DIS
LIN {X -0.020,Y -404.712,Z 1473.530,A 0.000,B 0.000,C 90.000,E1 275.454} C_DIS
LIN {X -0.092,Y -394.913,Z 1473.528,A 0.000,B 0.000,C 90.000,E1 274.992} C_DIS
LIN {X -0.164,Y -385.136,Z 1473.525,A 0.000,B 0.000,C 90.000,E1 274.588} C_DIS
LIN {X -0.077,Y -366.292,Z 1473.521,A 0.000,B 0.000,C 90.000,E1 273.841} C_DIS
LIN {X -0.131,Y -356.602,Z 1473.519,A 0.000,B 0.000,C 90.000,E1 273.498} C_DIS
LIN {X 0.082,Y -343.197,Z 1473.517,A 0.000,B 0.000,C 90.000,E1 273.037} C_DIS
LIN {X 0.143,Y -332.541,Z 1473.515,A 0.000,B 0.000,C 90.000,E1 272.751} C_DIS
LIN {X 0.138,Y -321.371,Z 1473.514,A 0.000,B 0.000,C 90.000,E1 272.522} C_DIS
LIN {X 0.020,Y -309.186,Z 1473.513,A 0.000,B 0.000,C 90.000,E1 272.350} C_DIS
LIN {X 0.051,Y -296.996,Z 1473.512,A 0.000,B 0.000,C 90.000,E1 272.236} C_DIS
LIN {X -0.047,Y -292.683,Z 1473.512,A 0.000,B 0.000,C 90.000,E1 272.236} C_DIS
LIN {X -0.060,Y -181.228,Z 1473.512,A 0.000,B 0.000,C 90.000,E1 272.236} C_DIS
LIN {X 0.081,Y -181.567,Z 1473.503,A 0.000,B 0.000,C 90.000,E1 270.458} C_DIS
LIN {X 0.070,Y -181.118,Z 1473.489,A 0.000,B 0.000,C 90.000,E1 267.936} C_DIS
LIN {X 0.058,Y -180.906,Z 1473.475,A 0.000,B 0.000,C 90.000,E1 265.412} C_DIS
LIN {X -0.065,Y -180.719,Z 1473.470,A 0.000,B 0.000,C 90.000,E1 264.609} C_DIS
LIN {X 0.033,Y -178.806,Z 1473.442,A 0.000,B 0.000,C 90.000,E1 259.511} C_DIS
LIN {X -0.060,Y -175.851,Z 1473.413,A 0.000,B 0.000,C 90.000,E1 254.448} C_DIS
LIN {X -0.078,Y -173.177,Z 1473.395,A 0.000,B 0.000,C 90.000,E1 251.040} C_DIS
LIN {X -0.075,Y -171.478,Z 1473.380,A 0.000,B 0.000,C 90.000,E1 248.465} C_DIS
LIN {X -0.087,Y -167.708,Z 1473.356,A 0.000,B 0.000,C 90.000,E1 244.152} C_DIS
LIN {X 0.076,Y -166.396,Z 1473.347,A 0.000,B 0.000,C 90.000,E1 242.359} C_DIS
LIN {X 0.068,Y -163.122,Z 1473.327,A 0.000,B 0.000,C 90.000,E1 238.869} C_DIS
LIN {X -0.106,Y -161.072,Z 1473.313,A 0.000,B 0.000,C 90.000,E1 236.294} C_DIS
LIN {X 0.005,Y -157.805,Z 1473.293,A 0.000,B 0.000,C 90.000,E1 232.718} C_DIS
LIN {X -0.057,Y -155.840,Z 1473.278,A 0.000,B 0.000,C 90.000,E1 230.070} C_DIS
LIN {X -0.001,Y -152.091,Z 1473.253,A 0.000,B 0.000,C 90.000,E1 225.567} C_DIS
LIN {X 0.018,Y -150.341,Z 1473.238,A 0.000,B 0.000,C 90.000,E1 222.852} C_DIS
LIN {X 0.039,Y -147.079,Z 1473.213,A 0.000,B 0.000,C 90.000,E1 218.302} C_DIS
LIN {X -0.057,Y -145.652,Z 1473.198,A 0.000,B 0.000,C 90.000,E1 215.598} C_DIS
LIN {X -0.053,Y -143.034,Z 1473.172,A 0.000,B 0.000,C 90.000,E1 211.003} C_DIS
LIN {X 0.073,Y -141.660,Z 1473.152,A 0.000,B 0.000,C 90.000,E1 207.257} C_DIS
LIN {X -0.007,Y -139.448,Z 1473.115,A 0.000,B 0.000,C 90.000,E1 200.791} C_DIS
LIN {X 0.044,Y -139.181,Z 1473.105,A 0.000,B 0.000,C 90.000,E1 198.906} C_DIS
LIN {X -0.063,Y -138.321,Z 1473.053,A 0.000,B 0.000,C 90.000,E1 189.613} C_DIS
LIN {X -0.057,Y -139.465,Z 1473.007,A 0.000,B 0.000,C 90.000,E1 181.203} C_DIS
LIN {X 0.023,Y -141.027,Z 1472.975,A 0.000,B 0.000,C 90.000,E1 175.584} C_DIS
LIN {X -0.022,Y -142.393,Z 1472.960,A 0.000,B 0.000,C 90.000,E1 172.818} C_DIS
LIN {X 0.041,Y -144.624,Z 1472.934,A 0.000,B 0.000,C 90.000,E1 168.173} C_DIS
LIN {X -0.040,Y -147.819,Z 1472.909,A 0.000,B 0.000,C 90.000,E1 163.614} C_DIS
LIN {X 0.047,Y -150.509,Z 1472.889,A 0.000,B 0.000,C 90.000,E1 159.934} C_DIS
LIN {X -0.074,Y -153.969,Z 1472.869,A 0.000,B 0.000,C 90.000,E1 156.357} C_DIS
LIN {X -0.012,Y -157.382,Z 1472.849,A 0.000,B 0.000,C 90.000,E1 152.743} C_DIS
LIN {X -0.070,Y -161.584,Z 1472.829,A 0.000,B 0.000,C 90.000,E1 149.203} C_DIS
LIN {X -0.059,Y -165.782,Z 1472.809,A 0.000,B 0.000,C 90.000,E1 145.674} C_DIS
LIN {X -0.074,Y -170.742,Z 1472.790,A 0.000,B 0.000,C 90.000,E1 142.190} C_DIS
LIN {X 0.085,Y -175.615,Z 1472.771,A 0.000,B 0.000,C 90.000,E1 138.690} C_DIS
LIN {X -0.045,Y -181.230,Z 1472.752,A 0.000,B 0.000,C 90.000,E1 135.324} C_DIS
LIN {X 0.086,Y -186.698,Z 1472.733,A 0.000,B 0.000,C 90.000,E1 131.919} C_DIS
LIN {X 0.037,Y -191.299,Z 1472.719,A 0.000,B 0.000,C 90.000,E1 129.439} C_DIS
LIN {X -0.032,Y -197.127,Z 1472.701,A 0.000,B 0.000,C 90.000,E1 126.171} C_DIS
LIN {X 0.035,Y -201.140,Z 1472.690,A 0.000,B 0.000,C 90.000,E1 124.119} C_DIS
LIN {X 0.020,Y -313.703,Z 1472.690,A 0.000,B 0.000,C 90.000,E1 124.119} C_DIS
LIN {X 0.043,Y -319.550,Z 1472.688,A 0.000,B 0.000,C 90.000,E1 123.913} C_DIS
LIN {X 0.100,Y -322.112,Z 1472.687,A 0.000,B 0.000,C 90.000,E1 123.706} C_DIS
LIN {X -0.114,Y -325.920,Z 1472.685,A 0.000,B 0.000,C 90.000,E1 123.293} C_DIS
LIN {X -0.006,Y -327.762,Z 1472.683,A 0.000,B 0.000,C 90.000,E1 122.959} C_DIS
LIN {X 0.104,Y -329.197,Z 1472.681,A 0.000,B 0.000,C 90.000,E1 122.625} C_DIS
LIN {X -0.120,Y -341.247,Z 1472.664,A 0.000,B 0.000,C 90.000,E1 119.539} C_DIS
LIN {X 0.114,Y -353.505,Z 1472.649,A 0.000,B 0.000,C 90.000,E1 116.744} C_DIS
LIN {X -0.099,Y -367.244,Z 1472.634,A 0.000,B 0.000,C 90.000,E1 114.079} C_DIS
LIN {X -0.005,Y -380.794,Z 1472.621,A 0.000,B 0.000,C 90.000,E1 111.716} C_DIS
LIN {X 0.160,Y -395.698,Z 1472.608,A 0.000,B 0.000,C 90.000,E1 109.396} C_DIS
LIN {X 0.068,Y -412.063,Z 1472.595,A 0.000,B 0.000,C 90.000,E1 107.166} C_DIS
LIN {X -0.156,Y -430.001,Z 1472.583,A 0.000,B 0.000,C 90.000,E1 105.009} C_DIS
LIN {X -0.072,Y -449.495,Z 1472.572,A 0.000,B 0.000,C 90.000,E1 102.883} C_DIS
LIN {X 0.191,Y -469.722,Z 1472.561,A 0.000,B 0.000,C 90.000,E1 100.894} C_DIS
LIN {X 0.133,Y -487.836,Z 1472.552,A 0.000,B 0.000,C 90.000,E1 99.321} C_DIS
LIN {X 0.206,Y -490.084,Z 1472.551,A 0.000,B 0.000,C 90.000,E1 99.095} C_DIS
LIN {X 0.176,Y -491.926,Z 1472.549,A 0.000,B 0.000,C 90.000,E1 98.859} C_DIS
LIN {X 0.145,Y -493.316,Z 1472.548,A 0.000,B 0.000,C 90.000,E1 98.624} C_DIS
LIN {X -0.111,Y -495.136,Z 1472.545,A 0.000,B 0.000,C 90.000,E1 98.163} C_DIS
LIN {X 0.132,Y -495.839,Z 1472.543,A 0.000,B 0.000,C 90.000,E1 97.644} C_DIS
LIN {X -0.105,Y -495.545,Z 1472.540,A 0.000,B 0.000,C 90.000,E1 97.182} C_DIS
LIN {X 0.154,Y -494.212,Z 1472.537,A 0.000,B 0.000,C 90.000,E1 96.663} C_DIS
LIN {X 0.066,Y -493.088,Z 1472.536,A 0.000,B 0.000,C 90.000,E1 96.429} C_DIS
LIN {X -0.177,Y -489.837,Z 1472.533,A 0.000,B 0.000,C 90.000,E1 95.967} C_DIS
LIN {X -0.074,Y -480.051,Z 1472.525,A 0.000,B 0.000,C 90.000,E1 94.473} C_DIS
LIN {X 0.146,Y -469.445,Z 1472.515,A 0.000,B 0.000,C 90.000,E1 92.694} C_DIS
LIN {X 0.086,Y -461.290,Z 1472.508,A 0.000,B 0.000,C 90.000,E1 91.432} C_DIS
LIN {X 0.127,Y -451.060,Z 1472.500,A 0.000,B 0.000,C 90.000,E1 89.885} C_DIS
LIN {X -0.077,Y -437.380,Z 1472.488,A 0.000,B 0.000,C 90.000,E1 87.822} C_DIS
LIN {X 0.137,Y -425.412,Z 1472.478,A 0.000,B 0.000,C 90.000,E1 85.931} C_DIS
LIN {X -0.139,Y -411.671,Z 1472.465,A 0.000,B 0.000,C 90.000,E1 83.799} C_DIS
LIN {X -0.085,Y -403.003,Z 1472.458,A 0.000,B 0.000,C 90.000,E1 82.413} C_DIS
LIN {X -0.021,Y -390.794,Z 1472.447,A 0.000,B 0.000,C 90.000,E1 80.443} C_DIS
LIN {X -0.096,Y -373.888,Z 1472.431,A 0.000,B 0.000,C 90.000,E1 77.589} C_DIS
LIN {X -0.003,Y -360.833,Z 1472.418,A 0.000,B 0.000,C 90.000,E1 75.227} C_DIS
LIN {X -0.064,Y -349.536,Z 1472.406,A 0.000,B 0.000,C 90.000,E1 73.142} C_DIS
LIN {X 0.068,Y -338.232,Z 1472.394,A 0.000,B 0.000,C 90.000,E1 70.986} C_DIS
LIN {X -0.097,Y -323.981,Z 1472.379,A 0.000,B 0.000,C 90.000,E1 68.209} C_DIS
LIN {X 0.036,Y -307.642,Z 1472.359,A 0.000,B 0.000,C 90.000,E1 64.665} C_DIS
LIN {X -0.009,Y -293.921,Z 1472.341,A 0.000,B 0.000,C 90.000,E1 61.385} C_DIS
LIN {X 0.124,Y -282.408,Z 1472.324,A 0.000,B 0.000,C 90.000,E1 58.329} C_DIS
LIN {X 0.061,Y -272.659,Z 1472.309,A 0.000,B 0.000,C 90.000,E1 55.595} C_DIS
LIN {X -0.087,Y -262.028,Z 1472.291,A 0.000,B 0.000,C 90.000,E1 52.477} C_DIS
LIN {X 0.139,Y -250.911,Z 1472.272,A 0.000,B 0.000,C 90.000,E1 48.852} C_DIS
LIN {X -0.022,Y -240.730,Z 1472.251,A 0.000,B 0.000,C 90.000,E1 45.243} C_DIS
LIN {X 0.017,Y -231.626,Z 1472.231,A 0.000,B 0.000,C 90.000,E1 41.515} C_DIS
LIN {X 0.008,Y -223.599,Z 1472.210,A 0.000,B 0.000,C 90.000,E1 37.729} C_DIS
LIN {X 0.063,Y -216.555,Z 1472.188,A 0.000,B 0.000,C 90.000,E1 33.865} C_DIS
LIN {X -0.093,Y -210.260,Z 1472.167,A 0.000,B 0.000,C 90.000,E1 30.001} C_DIS
LIN {X -0.034,Y -204.863,Z 1472.145,A 0.000,B 0.000,C 90.000,E1 26.027} C_DIS
LIN {X -0.036,Y -200.170,Z 1472.122,A 0.000,B 0.000,C 90.000,E1 22.025} C_DIS
LIN {X -0.026,Y -195.516,Z 1472.095,A 0.000,B 0.000,C 90.000,E1 17.166} C_DIS
LIN {X 0.040,Y -191.927,Z 1472.068,A 0.000,B 0.000,C 90.000,E1 12.243} C_DIS
LIN {X 0.009,Y -189.080,Z 1472.036,A 0.000,B 0.000,C 90.000,E1 6.486} C_DIS
LIN {X -0.034,Y -187.437,Z 1471.997,A 0.000,B 0.000,C 90.000,E1 359.542} C_DIS
LIN {X 0.006,Y -187.443,Z 1471.970,A 0.000,B 0.000,C 90.000,E1 354.546} C_DIS
LIN {X 0.063,Y -189.146,Z 1471.928,A 0.000,B 0.000,C 90.000,E1 347.061} C_DIS
LIN {X 0.081,Y -192.193,Z 1471.896,A 0.000,B 0.000,C 90.000,E1 341.275} C_DIS
LIN {X 0.075,Y -196.061,Z 1471.869,A 0.000,B 0.000,C 90.000,E1 336.357} C_DIS
LIN {X 0.019,Y -200.333,Z 1471.846,A 0.000,B 0.000,C 90.000,E1 332.308} C_DIS
LIN {X 0.029,Y -205.679,Z 1471.824,A 0.000,B 0.000,C 90.000,E1 328.280} C_DIS
LIN {X 0.003,Y -210.953,Z 1471.806,A 0.000,B 0.000,C 90.000,E1 325.102} C_DIS
LIN {X -0.116,Y -217.011,Z 1471.789,A 0.000,B 0.000,C 90.000,E1 321.984} C_DIS
LIN {X -0.022,Y -224.085,Z 1471.771,A 0.000,B 0.000,C 90.000,E1 318.852} C_DIS
LIN {X -0.096,Y -232.041,Z 1471.754,A 0.000,B 0.000,C 90.000,E1 315.810} C_DIS
LIN {X 0.030,Y -242.154,Z 1471.736,A 0.000,B 0.000,C 90.000,E1 312.405} C_DIS
LIN {X -0.064,Y -250.959,Z 1471.721,A 0.000,B 0.000,C 90.000,E1 309.850} C_DIS
LIN {X -0.015,Y -262.396,Z 1471.705,A 0.000,B 0.000,C 90.000,E1 306.950} C_DIS
LIN {X -0.044,Y -270.310,Z 1471.695,A 0.000,B 0.000,C 90.000,E1 305.185} C_DIS
LIN {X -0.041,Y -277.305,Z 1471.688,A 0.000,B 0.000,C 90.000,E1 303.785} C_DIS
LIN {X -0.059,Y -291.076,Z 1471.674,A 0.000,B 0.000,C 90.000,E1 301.386} C_DIS
LIN {X 0.159,Y -301.863,Z 1471.665,A 0.000,B 0.000,C 90.000,E1 299.667} C_DIS
LIN {X -0.152,Y -310.979,Z 1471.658,A 0.000,B 0.000,C 90.000,E1 298.487} C_DIS
LIN {X -0.164,Y -321.291,Z 1471.651,A 0.000,B 0.000,C 90.000,E1 297.257} C_DIS
LIN {X 0.014,Y -340.178,Z 1471.640,A 0.000,B 0.000,C 90.000,E1 295.207} C_DIS
LIN {X -0.062,Y -356.650,Z 1471.631,A 0.000,B 0.000,C 90.000,E1 293.567} C_DIS
LIN {X 0.026,Y -367.453,Z 1471.625,A 0.000,B 0.000,C 90.000,E1 292.461} C_DIS
LIN {X 0.086,Y -377.994,Z 1471.619,A 0.000,B 0.000,C 90.000,E1 291.354} C_DIS
LIN {X -0.069,Y -390.930,Z 1471.611,A 0.000,B 0.000,C 90.000,E1 289.993} C_DIS
LIN {X -0.179,Y -403.464,Z 1471.603,A 0.000,B 0.000,C 90.000,E1 288.598} C_DIS
LIN {X 0.005,Y -412.914,Z 1471.597,A 0.000,B 0.000,C 90.000,E1 287.457} C_DIS
LIN {X 0.068,Y -419.422,Z 1471.592,A 0.000,B 0.000,C 90.000,E1 286.622} C_DIS
LIN {X -0.220,Y -425.306,Z 1471.588,A 0.000,B 0.000,C 90.000,E1 285.843} C_DIS
LIN {X 0.203,Y -428.822,Z 1471.585,A 0.000,B 0.000,C 90.000,E1 285.245} C_DIS
LIN {X 0.126,Y -431.943,Z 1471.582,A 0.000,B 0.000,C 90.000,E1 284.717} C_DIS
LIN {X -0.056,Y -435.889,Z 1471.577,A 0.000,B 0.000,C 90.000,E1 283.939} C_DIS
LIN {X 0.111,Y -439.137,Z 1471.573,A 0.000,B 0.000,C 90.000,E1 283.119} C_DIS
LIN {X 0.100,Y -440.871,Z 1471.570,A 0.000,B 0.000,C 90.000,E1 282.591} C_DIS
LIN {X 0.096,Y -442.245,Z 1471.567,A 0.000,B 0.000,C 90.000,E1 282.063} C_DIS
LIN {X 0.100,Y -443.210,Z 1471.564,A 0.000,B 0.000,C 90.000,E1 281.535} C_DIS
LIN {X 0.111,Y -443.706,Z 1471.561,A 0.000,B 0.000,C 90.000,E1 281.007} C_DIS
LIN {X 0.045,Y -443.756,Z 1471.558,A 0.000,B 0.000,C 90.000,E1 280.489} C_DIS
LIN {X 0.064,Y -443.248,Z 1471.555,A 0.000,B 0.000,C 90.000,E1 279.962} C_DIS
LIN {X 0.007,Y -442.198,Z 1471.552,A 0.000,B 0.000,C 90.000,E1 279.443} C_DIS
LIN {X 0.020,Y -440.508,Z 1471.550,A 0.000,B 0.000,C 90.000,E1 278.916} C_DIS
LIN {X -0.042,Y -438.074,Z 1471.547,A 0.000,B 0.000,C 90.000,E1 278.398} C_DIS
LIN {X 0.167,Y -436.628,Z 1471.545,A 0.000,B 0.000,C 90.000,E1 278.106} C_DIS
LIN {X 0.082,Y -432.878,Z 1471.542,A 0.000,B 0.000,C 90.000,E1 277.587} C_DIS
LIN {X -0.018,Y -428.089,Z 1471.539,A 0.000,B 0.000,C 90.000,E1 277.068} C_DIS
LIN {X 0.026,Y -422.335,Z 1471.536,A 0.000,B 0.000,C 90.000,E1 276.549} C_DIS
LIN {X 0.020,Y -416.053,Z 1471.534,A 0.000,B 0.000,C 90.000,E1 276.087} C_DIS
LIN {X 0.004,Y -409.636,Z 1471.532,A 0.000,B 0.000,C 90.000,E1 275.682} C_DIS
LIN {X -0.055,Y -403.034,Z 1471.530,A 0.000,B 0.000,C 90.000,E1 275.334} C_DIS
LIN {X -0.092,Y -393.150,Z 1471.527,A 0.000,B 0.000,C 90.000,E1 274.878} C_DIS
LIN {X -0.080,Y -383.368,Z 1471.525,A 0.000,B 0.000,C 90.000,E1 274.473} C_DIS
LIN {X 0.032,Y -364.484,Z 1471.521,A 0.000,B 0.000,C 90.000,E1 273.726} C_DIS
LIN {X -0.023,Y -354.556,Z 1471.519,A 0.000,B 0.000,C 90.000,E1 273.383} C_DIS
LIN {X 0.174,Y -344.387,Z 1471.517,A 0.000,B 0.000,C 90.000,E1 273.037} C_DIS
LIN {X -0.118,Y -333.804,Z 1471.516,A 0.000,B 0.000,C 90.000,E1 272.808} C_DIS
LIN {X -0.103,Y -322.831,Z 1471.514,A 0.000,B 0.000,C 90.000,E1 272.579} C_DIS
LIN {X 0.124,Y -315.301,Z 1471.514,A 0.000,B 0.000,C 90.000,E1 272.407} C_DIS
LIN {X 0.117,Y -306.402,Z 1471.513,A 0.000,B 0.000,C 90.000,E1 272.293} C_DIS
LIN {X 0.030,Y -296.560,Z 1471.512,A 0.000,B 0.000,C 90.000,E1 272.236} C_DIS
LIN {X -0.073,Y -290.070,Z 1471.512,A 0.000,B 0.000,C 90.000,E1 272.236} C_DIS
LIN {X -0.079,Y -181.229,Z 1471.512,A 0.000,B 0.000,C 90.000,E1 272.236} C_DIS
LIN {X -0.064,Y -181.566,Z 1471.503,A 0.000,B 0.000,C 90.000,E1 270.516} C_DIS
LIN {X -0.074,Y -181.120,Z 1471.489,A 0.000,B 0.000,C 90.000,E1 267.993} C_DIS
LIN {X -0.085,Y -180.906,Z 1471.475,A 0.000,B 0.000,C 90.000,E1 265.469} C_DIS
LIN {X -0.029,Y -180.724,Z 1471.470,A 0.000,B 0.000,C 90.000,E1 264.609} C_DIS
LIN {X 0.069,Y -178.813,Z 1471.442,A 0.000,B 0.000,C 90.000,E1 259.511} C_DIS
LIN {X -0.025,Y -175.857,Z 1471.414,A 0.000,B 0.000,C 90.000,E1 254.448} C_DIS
LIN {X -0.042,Y -173.185,Z 1471.395,A 0.000,B 0.000,C 90.000,E1 251.040} C_DIS
LIN {X -0.040,Y -171.488,Z 1471.380,A 0.000,B 0.000,C 90.000,E1 248.465} C_DIS
LIN {X -0.052,Y -167.717,Z 1471.356,A 0.000,B 0.000,C 90.000,E1 244.152} C_DIS
LIN {X -0.036,Y -166.409,Z 1471.347,A 0.000,B 0.000,C 90.000,E1 242.410} C_DIS
LIN {X -0.038,Y -163.132,Z 1471.327,A 0.000,B 0.000,C 90.000,E1 238.918} C_DIS
LIN {X -0.072,Y -161.085,Z 1471.313,A 0.000,B 0.000,C 90.000,E1 236.294} C_DIS
LIN {X 0.038,Y -157.815,Z 1471.293,A 0.000,B 0.000,C 90.000,E1 232.718} C_DIS
LIN {X -0.024,Y -155.849,Z 1471.278,A 0.000,B 0.000,C 90.000,E1 230.070} C_DIS
LIN {X 0.032,Y -152.099,Z 1471.253,A 0.000,B 0.000,C 90.000,E1 225.567} C_DIS
LIN {X 0.051,Y -150.350,Z 1471.238,A 0.000,B 0.000,C 90.000,E1 222.852} C_DIS
LIN {X -0.020,Y -147.087,Z 1471.213,A 0.000,B 0.000,C 90.000,E1 218.338} C_DIS
LIN {X -0.025,Y -145.659,Z 1471.198,A 0.000,B 0.000,C 90.000,E1 215.598} C_DIS
LIN {X -0.022,Y -143.040,Z 1471.172,A 0.000,B 0.000,C 90.000,E1 211.003} C_DIS
LIN {X -0.021,Y -141.665,Z 1471.152,A 0.000,B 0.000,C 90.000,E1 207.308} C_DIS
LIN {X 0.023,Y -139.450,Z 1471.116,A 0.000,B 0.000,C 90.000,E1 200.791} C_DIS
LIN {X -0.055,Y -139.184,Z 1471.105,A 0.000,B 0.000,C 90.000,E1 198.960} C_DIS
LIN {X -0.033,Y -138.321,Z 1471.053,A 0.000,B 0.000,C 90.000,E1 189.613} C_DIS
LIN {X -0.026,Y -139.462,Z 1471.007,A 0.000,B 0.000,C 90.000,E1 181.203} C_DIS
LIN {X 0.055,Y -141.021,Z 1470.976,A 0.000,B 0.000,C 90.000,E1 175.584} C_DIS
LIN {X 0.009,Y -142.386,Z 1470.960,A 0.000,B 0.000,C 90.000,E1 172.818} C_DIS
LIN {X -0.070,Y -144.616,Z 1470.934,A 0.000,B 0.000,C 90.000,E1 168.229} C_DIS
LIN {X -0.008,Y -147.811,Z 1470.909,A 0.000,B 0.000,C 90.000,E1 163.614} C_DIS
LIN {X 0.079,Y -150.499,Z 1470.889,A 0.000,B 0.000,C 90.000,E1 159.934} C_DIS
LIN {X -0.041,Y -153.957,Z 1470.869,A 0.000,B 0.000,C 90.000,E1 156.357} C_DIS
LIN {X 0.021,Y -157.369,Z 1470.849,A 0.000,B 0.000,C 90.000,E1 152.743} C_DIS
LIN {X -0.036,Y -161.568,Z 1470.829,A 0.000,B 0.000,C 90.000,E1 149.203} C_DIS
LIN {X -0.025,Y -165.766,Z 1470.809,A 0.000,B 0.000,C 90.000,E1 145.674} C_DIS
LIN {X -0.039,Y -170.724,Z 1470.790,A 0.000,B 0.000,C 90.000,E1 142.190} C_DIS
LIN {X 0.005,Y -175.596,Z 1470.771,A 0.000,B 0.000,C 90.000,E1 138.728} C_DIS
LIN {X -0.008,Y -181.213,Z 1470.752,A 0.000,B 0.000,C 90.000,E1 135.324} C_DIS
LIN {X -0.016,Y -186.678,Z 1470.733,A 0.000,B 0.000,C 90.000,E1 131.962} C_DIS
LIN {X -0.073,Y -191.280,Z 1470.719,A 0.000,B 0.000,C 90.000,E1 129.483} C_DIS
LIN {X 0.007,Y -197.106,Z 1470.701,A 0.000,B 0.000,C 90.000,E1 126.171} C_DIS
LIN {X 0.026,Y -201.090,Z 1470.690,A 0.000,B 0.000,C 90.000,E1 124.151} C_DIS
LIN {X 0.182,Y -313.106,Z 1470.690,A 0.000,B 0.000,C 90.000,E1 124.119} C_DIS
LIN {X 0.049,Y -315.092,Z 1470.690,A 0.000,B 0.000,C 90.000,E1 124.119} C_DIS
LIN {X 0.105,Y -319.687,Z 1470.688,A 0.000,B 0.000,C 90.000,E1 123.913} C_DIS
LIN {X 0.162,Y -322.172,Z 1470.687,A 0.000,B 0.000,C 90.000,E1 123.706} C_DIS
LIN {X -0.119,Y -325.987,Z 1470.685,A 0.000,B 0.000,C 90.000,E1 123.293} C_DIS
LIN {X -0.030,Y -327.804,Z 1470.683,A 0.000,B 0.000,C 90.000,E1 122.959} C_DIS
LIN {X 0.062,Y -329.216,Z 1470.681,A 0.000,B 0.000,C 90.000,E1 122.625} C_DIS
LIN {X -0.164,Y -341.257,Z 1470.664,A 0.000,B 0.000,C 90.000,E1 119.539} C_DIS
LIN {X 0.068,Y -353.518,Z 1470.649,A 0.000,B 0.000,C 90.000,E1 116.744} C_DIS
LIN {X -0.145,Y -367.261,Z 1470.634,A 0.000,B 0.000,C 90.000,E1 114.079} C_DIS
LIN {X -0.053,Y -380.814,Z 1470.621,A 0.000,B 0.000,C 90.000,E1 111.716} C_DIS
LIN {X 0.110,Y -395.722,Z 1470.608,A 0.000,B 0.000,C 90.000,E1 109.396} C_DIS
LIN {X 0.017,Y -412.091,Z 1470.595,A 0.000,B 0.000,C 90.000,E1 107.166} C_DIS
LIN {X -0.209,Y -430.033,Z 1470.583,A 0.000,B 0.000,C 90.000,E1 105.009} C_DIS
LIN {X -0.125,Y -449.532,Z 1470.572,A 0.000,B 0.000,C 90.000,E1 102.883} C_DIS
LIN {X 0.139,Y -469.761,Z 1470.561,A 0.000,B 0.000,C 90.000,E1 100.894} C_DIS
LIN {X 0.083,Y -487.875,Z 1470.552,A 0.000,B 0.000,C 90.000,E1 99.321} C_DIS
LIN {X 0.155,Y -490.083,Z 1470.551,A 0.000,B 0.000,C 90.000,E1 99.095} C_DIS
LIN {X 0.104,Y -491.913,Z 1470.549,A 0.000,B 0.000,C 90.000,E1 98.859} C_DIS
LIN {X 0.051,Y -493.291,Z 1470.548,A 0.000,B 0.000,C 90.000,E1 98.624} C_DIS
LIN {X -0.205,Y -495.067,Z 1470.545,A 0.000,B 0.000,C 90.000,E1 98.163} C_DIS
LIN {X 0.037,Y -495.733,Z 1470.542,A 0.000,B 0.000,C 90.000,E1 97.644} C_DIS
LIN {X -0.200,Y -495.404,Z 1470.540,A 0.000,B 0.000,C 90.000,E1 97.182} C_DIS
LIN {X 0.059,Y -494.032,Z 1470.537,A 0.000,B 0.000,C 90.000,E1 96.663} C_DIS
LIN {X -0.031,Y -492.883,Z 1470.536,A 0.000,B 0.000,C 90.000,E1 96.429} C_DIS
LIN {X 0.215,Y -489.605,Z 1470.533,A 0.000,B 0.000,C 90.000,E1 95.910} C_DIS
LIN {X -0.173,Y -479.817,Z 1470.525,A 0.000,B 0.000,C 90.000,E1 94.473} C_DIS
LIN {X 0.045,Y -469.198,Z 1470.515,A 0.000,B 0.000,C 90.000,E1 92.694} C_DIS
LIN {X -0.016,Y -461.043,Z 1470.508,A 0.000,B 0.000,C 90.000,E1 91.432} C_DIS
LIN {X 0.023,Y -450.806,Z 1470.499,A 0.000,B 0.000,C 90.000,E1 89.885} C_DIS
LIN {X -0.184,Y -437.184,Z 1470.488,A 0.000,B 0.000,C 90.000,E1 87.822} C_DIS
LIN {X -0.104,Y -426.946,Z 1470.479,A 0.000,B 0.000,C 90.000,E1 86.216} C_DIS
LIN {X -0.048,Y -414.959,Z 1470.468,A 0.000,B 0.000,C 90.000,E1 84.318} C_DIS
LIN {X 0.109,Y -404.673,Z 1470.459,A 0.000,B 0.000,C 90.000,E1 82.648} C_DIS
LIN {X -0.127,Y -390.745,Z 1470.447,A 0.000,B 0.000,C 90.000,E1 80.443} C_DIS
LIN {X -0.198,Y -373.837,Z 1470.431,A 0.000,B 0.000,C 90.000,E1 77.589} C_DIS
LIN {X -0.103,Y -360.808,Z 1470.418,A 0.000,B 0.000,C 90.000,E1 75.227} C_DIS
LIN {X -0.161,Y -349.495,Z 1470.406,A 0.000,B 0.000,C 90.000,E1 73.142} C_DIS
LIN {X 0.082,Y -338.170,Z 1470.394,A 0.000,B 0.000,C 90.000,E1 70.967} C_DIS
LIN {X 0.111,Y -323.933,Z 1470.379,A 0.000,B 0.000,C 90.000,E1 68.156} C_DIS
LIN {X -0.053,Y -307.592,Z 1470.359,A 0.000,B 0.000,C 90.000,E1 64.665} C_DIS
LIN {X -0.097,Y -293.850,Z 1470.341,A 0.000,B 0.000,C 90.000,E1 61.385} C_DIS
LIN {X 0.039,Y -282.328,Z 1470.324,A 0.000,B 0.000,C 90.000,E1 58.329} C_DIS
LIN {X -0.023,Y -272.590,Z 1470.309,A 0.000,B 0.000,C 90.000,E1 55.595} C_DIS
LIN {X 0.038,Y -261.993,Z 1470.291,A 0.000,B 0.000,C 90.000,E1 52.431} C_DIS
LIN {X 0.059,Y -250.933,Z 1470.271,A 0.000,B 0.000,C 90.000,E1 48.852} C_DIS
LIN {X -0.097,Y -240.818,Z 1470.251,A 0.000,B 0.000,C 90.000,E1 45.243} C_DIS
LIN {X -0.053,Y -231.752,Z 1470.231,A 0.000,B 0.000,C 90.000,E1 41.515} C_DIS
LIN {X -0.055,Y -223.759,Z 1470.209,A 0.000,B 0.000,C 90.000,E1 37.729} C_DIS
LIN {X 0.007,Y -216.729,Z 1470.188,A 0.000,B 0.000,C 90.000,E1 33.865} C_DIS
LIN {X 0.040,Y -210.463,Z 1470.167,A 0.000,B 0.000,C 90.000,E1 29.951} C_DIS
LIN {X 0.108,Y -205.072,Z 1470.145,A 0.000,B 0.000,C 90.000,E1 25.976} C_DIS
LIN {X -0.071,Y -200.386,Z 1470.122,A 0.000,B 0.000,C 90.000,E1 22.025} C_DIS
LIN {X 0.006,Y -195.746,Z 1470.095,A 0.000,B 0.000,C 90.000,E1 17.149} C_DIS
LIN {X 0.023,Y -192.170,Z 1470.068,A 0.000,B 0.000,C 90.000,E1 12.243} C_DIS
LIN {X -0.073,Y -189.041,Z 1470.031,A 0.000,B 0.000,C 90.000,E1 5.682} C_DIS
LIN {X -0.034,Y -187.716,Z 1469.997,A 0.000,B 0.000,C 90.000,E1 359.542} C_DIS
LIN {X 0.016,Y -187.701,Z 1469.970,A 0.000,B 0.000,C 90.000,E1 354.546} C_DIS
LIN {X -0.097,Y -189.367,Z 1469.928,A 0.000,B 0.000,C 90.000,E1 347.117} C_DIS
LIN {X -0.068,Y -192.377,Z 1469.896,A 0.000,B 0.000,C 90.000,E1 341.329} C_DIS
LIN {X -0.064,Y -196.219,Z 1469.869,A 0.000,B 0.000,C 90.000,E1 336.410} C_DIS
LIN {X -0.111,Y -200.462,Z 1469.846,A 0.000,B 0.000,C 90.000,E1 332.359} C_DIS
LIN {X -0.094,Y -205.809,Z 1469.824,A 0.000,B 0.000,C 90.000,E1 328.329} C_DIS
LIN {X 0.059,Y -211.079,Z 1469.806,A 0.000,B 0.000,C 90.000,E1 325.102} C_DIS
LIN {X -0.054,Y -217.162,Z 1469.789,A 0.000,B 0.000,C 90.000,E1 321.984} C_DIS
LIN {X 0.045,Y -224.223,Z 1469.771,A 0.000,B 0.000,C 90.000,E1 318.852} C_DIS
LIN {X -0.023,Y -232.196,Z 1469.755,A 0.000,B 0.000,C 90.000,E1 315.810} C_DIS
LIN {X -0.067,Y -242.330,Z 1469.736,A 0.000,B 0.000,C 90.000,E1 312.447} C_DIS
LIN {X 0.037,Y -252.481,Z 1469.719,A 0.000,B 0.000,C 90.000,E1 309.483} C_DIS
LIN {X 0.026,Y -265.614,Z 1469.701,A 0.000,B 0.000,C 90.000,E1 306.251} C_DIS
LIN {X 0.052,Y -273.849,Z 1469.692,A 0.000,B 0.000,C 90.000,E1 304.485} C_DIS
LIN {X 0.101,Y -281.185,Z 1469.684,A 0.000,B 0.000,C 90.000,E1 303.086} C_DIS
LIN {X 0.037,Y -293.225,Z 1469.673,A 0.000,B 0.000,C 90.000,E1 301.052} C_DIS
LIN {X -0.133,Y -301.890,Z 1469.665,A 0.000,B 0.000,C 90.000,E1 299.745} C_DIS
LIN {X -0.135,Y -311.136,Z 1469.658,A 0.000,B 0.000,C 90.000,E1 298.487} C_DIS
LIN {X 0.024,Y -321.634,Z 1469.651,A 0.000,B 0.000,C 90.000,E1 297.206} C_DIS
LIN {X 0.020,Y -340.857,Z 1469.640,A 0.000,B 0.000,C 90.000,E1 295.155} C_DIS
LIN {X -0.075,Y -357.397,Z 1469.631,A 0.000,B 0.000,C 90.000,E1 293.515} C_DIS
LIN {X 0.020,Y -368.164,Z 1469.625,A 0.000,B 0.000,C 90.000,E1 292.408} C_DIS
LIN {X 0.179,Y -378.736,Z 1469.618,A 0.000,B 0.000,C 90.000,E1 291.280} C_DIS
LIN {X 0.041,Y -391.420,Z 1469.611,A 0.000,B 0.000,C 90.000,E1 289.939} C_DIS
LIN {X 0.056,Y -403.820,Z 1469.603,A 0.000,B 0.000,C 90.000,E1 288.544} C_DIS
LIN {X -0.141,Y -413.282,Z 1469.597,A 0.000,B 0.000,C 90.000,E1 287.457} C_DIS
LIN {X -0.076,Y -419.816,Z 1469.592,A 0.000,B 0.000,C 90.000,E1 286.622} C_DIS
LIN {X 0.046,Y -425.721,Z 1469.588,A 0.000,B 0.000,C 90.000,E1 285.788} C_DIS
LIN {X -0.185,Y -430.817,Z 1469.583,A 0.000,B 0.000,C 90.000,E1 285.009} C_DIS
LIN {X 0.038,Y -435.028,Z 1469.579,A 0.000,B 0.000,C 90.000,E1 284.175} C_DIS
LIN {X 0.200,Y -438.480,Z 1469.574,A 0.000,B 0.000,C 90.000,E1 283.355} C_DIS
LIN {X -0.034,Y -441.243,Z 1469.570,A 0.000,B 0.000,C 90.000,E1 282.591} C_DIS
LIN {X -0.037,Y -442.623,Z 1469.567,A 0.000,B 0.000,C 90.000,E1 282.063} C_DIS
LIN {X -0.030,Y -443.593,Z 1469.564,A 0.000,B 0.000,C 90.000,E1 281.535} C_DIS
LIN {X -0.017,Y -444.053,Z 1469.561,A 0.000,B 0.000,C 90.000,E1 281.007} C_DIS
LIN {X -0.081,Y -444.094,Z 1469.558,A 0.000,B 0.000,C 90.000,E1 280.489} C_DIS
LIN {X -0.061,Y -443.606,Z 1469.555,A 0.000,B 0.000,C 90.000,E1 279.962} C_DIS
LIN {X -0.116,Y -442.562,Z 1469.552,A 0.000,B 0.000,C 90.000,E1 279.443} C_DIS
LIN {X -0.100,Y -440.895,Z 1469.549,A 0.000,B 0.000,C 90.000,E1 278.916} C_DIS
LIN {X -0.159,Y -438.505,Z 1469.547,A 0.000,B 0.000,C 90.000,E1 278.398} C_DIS
LIN {X 0.051,Y -437.012,Z 1469.545,A 0.000,B 0.000,C 90.000,E1 278.106} C_DIS
LIN {X -0.030,Y -433.369,Z 1469.542,A 0.000,B 0.000,C 90.000,E1 277.587} C_DIS
LIN {X -0.127,Y -428.589,Z 1469.539,A 0.000,B 0.000,C 90.000,E1 277.068} C_DIS
LIN {X -0.070,Y -422.858,Z 1469.536,A 0.000,B 0.000,C 90.000,E1 276.549} C_DIS
LIN {X -0.045,Y -416.664,Z 1469.534,A 0.000,B 0.000,C 90.000,E1 276.087} C_DIS
LIN {X -0.048,Y -410.283,Z 1469.531,A 0.000,B 0.000,C 90.000,E1 275.682} C_DIS
LIN {X -0.059,Y -400.298,Z 1469.529,A 0.000,B 0.000,C 90.000,E1 275.163} C_DIS
LIN {X 0.111,Y -390.532,Z 1469.526,A 0.000,B 0.000,C 90.000,E1 274.702} C_DIS
LIN {X 0.078,Y -374.483,Z 1469.523,A 0.000,B 0.000,C 90.000,E1 274.073} C_DIS
LIN {X -0.022,Y -358.710,Z 1469.519,A 0.000,B 0.000,C 90.000,E1 273.498} C_DIS
LIN {X 0.048,Y -348.513,Z 1469.518,A 0.000,B 0.000,C 90.000,E1 273.154} C_DIS
LIN {X 0.085,Y -338.304,Z 1469.516,A 0.000,B 0.000,C 90.000,E1 272.865} C_DIS
LIN {X -0.001,Y -327.452,Z 1469.515,A 0.000,B 0.000,C 90.000,E1 272.636} C_DIS
LIN {X -0.142,Y -316.601,Z 1469.514,A 0.000,B 0.000,C 90.000,E1 272.465} C_DIS
LIN {X -0.146,Y -307.981,Z 1469.513,A 0.000,B 0.000,C 90.000,E1 272.350} C_DIS
LIN {X 0.064,Y -298.286,Z 1469.512,A 0.000,B 0.000,C 90.000,E1 272.236} C_DIS
LIN {X -0.045,Y -292.774,Z 1469.512,A 0.000,B 0.000,C 90.000,E1 272.236} C_DIS
LIN {X -0.062,Y -181.228,Z 1469.512,A 0.000,B 0.000,C 90.000,E1 272.236} C_DIS
LIN {X -0.049,Y -181.565,Z 1469.503,A 0.000,B 0.000,C 90.000,E1 270.516} C_DIS
LIN {X -0.060,Y -181.120,Z 1469.489,A 0.000,B 0.000,C 90.000,E1 267.993} C_DIS
LIN {X -0.071,Y -180.907,Z 1469.475,A 0.000,B 0.000,C 90.000,E1 265.469} C_DIS
LIN {X -0.014,Y -180.726,Z 1469.470,A 0.000,B 0.000,C 90.000,E1 264.609} C_DIS
LIN {X 0.083,Y -178.815,Z 1469.442,A 0.000,B 0.000,C 90.000,E1 259.511} C_DIS
LIN {X -0.010,Y -175.860,Z 1469.414,A 0.000,B 0.000,C 90.000,E1 254.448} C_DIS
LIN {X 0.039,Y -173.825,Z 1469.399,A 0.000,B 0.000,C 90.000,E1 251.873} C_DIS
LIN {X -0.026,Y -171.492,Z 1469.380,A 0.000,B 0.000,C 90.000,E1 248.465} C_DIS
LIN {X -0.038,Y -167.720,Z 1469.356,A 0.000,B 0.000,C 90.000,E1 244.152} C_DIS
LIN {X -0.023,Y -166.414,Z 1469.347,A 0.000,B 0.000,C 90.000,E1 242.410} C_DIS
LIN {X -0.024,Y -163.136,Z 1469.327,A 0.000,B 0.000,C 90.000,E1 238.918} C_DIS
LIN {X -0.059,Y -161.089,Z 1469.313,A 0.000,B 0.000,C 90.000,E1 236.294} C_DIS
LIN {X -0.074,Y -157.818,Z 1469.293,A 0.000,B 0.000,C 90.000,E1 232.763} C_DIS
LIN {X -0.011,Y -155.853,Z 1469.278,A 0.000,B 0.000,C 90.000,E1 230.070} C_DIS
LIN {X 0.046,Y -152.102,Z 1469.253,A 0.000,B 0.000,C 90.000,E1 225.567} C_DIS
LIN {X 0.064,Y -150.354,Z 1469.238,A 0.000,B 0.000,C 90.000,E1 222.852} C_DIS
LIN {X -0.008,Y -147.090,Z 1469.213,A 0.000,B 0.000,C 90.000,E1 218.338} C_DIS
LIN {X -0.013,Y -145.661,Z 1469.198,A 0.000,B 0.000,C 90.000,E1 215.598} C_DIS
LIN {X -0.010,Y -143.043,Z 1469.172,A 0.000,B 0.000,C 90.000,E1 211.003} C_DIS
LIN {X -0.009,Y -141.667,Z 1469.152,A 0.000,B 0.000,C 90.000,E1 207.308} C_DIS
LIN {X 0.036,Y -139.450,Z 1469.116,A 0.000,B 0.000,C 90.000,E1 200.791} C_DIS
LIN {X -0.043,Y -139.185,Z 1469.105,A 0.000,B 0.000,C 90.000,E1 198.960} C_DIS
LIN {X -0.020,Y -138.322,Z 1469.053,A 0.000,B 0.000,C 90.000,E1 189.613} C_DIS
LIN {X -0.013,Y -139.461,Z 1469.007,A 0.000,B 0.000,C 90.000,E1 181.203} C_DIS
LIN {X 0.068,Y -141.019,Z 1468.976,A 0.000,B 0.000,C 90.000,E1 175.584} C_DIS
LIN {X 0.022,Y -142.383,Z 1468.960,A 0.000,B 0.000,C 90.000,E1 172.818} C_DIS
LIN {X -0.056,Y -144.613,Z 1468.934,A 0.000,B 0.000,C 90.000,E1 168.229} C_DIS
LIN {X 0.004,Y -147.807,Z 1468.909,A 0.000,B 0.000,C 90.000,E1 163.614} C_DIS
LIN {X 0.041,Y -150.495,Z 1468.889,A 0.000,B 0.000,C 90.000,E1 159.953} C_DIS
LIN {X -0.028,Y -153.952,Z 1468.869,A 0.000,B 0.000,C 90.000,E1 156.357} C_DIS
LIN {X 0.035,Y -157.363,Z 1468.849,A 0.000,B 0.000,C 90.000,E1 152.743} C_DIS
LIN {X -0.022,Y -161.562,Z 1468.829,A 0.000,B 0.000,C 90.000,E1 149.203} C_DIS
LIN {X -0.011,Y -165.760,Z 1468.809,A 0.000,B 0.000,C 90.000,E1 145.674} C_DIS
LIN {X -0.024,Y -170.716,Z 1468.790,A 0.000,B 0.000,C 90.000,E1 142.190} C_DIS
LIN {X 0.019,Y -175.590,Z 1468.771,A 0.000,B 0.000,C 90.000,E1 138.728} C_DIS
LIN {X 0.006,Y -181.206,Z 1468.752,A 0.000,B 0.000,C 90.000,E1 135.324} C_DIS
LIN {X -0.001,Y -186.670,Z 1468.733,A 0.000,B 0.000,C 90.000,E1 131.962} C_DIS
LIN {X -0.058,Y -191.273,Z 1468.719,A 0.000,B 0.000,C 90.000,E1 129.483} C_DIS
LIN {X 0.023,Y -197.096,Z 1468.701,A 0.000,B 0.000,C 90.000,E1 126.171} C_DIS
LIN {X -0.060,Y -201.051,Z 1468.690,A 0.000,B 0.000,C 90.000,E1 124.199} C_DIS
LIN {X -0.127,Y -313.452,Z 1468.690,A 0.000,B 0.000,C 90.000,E1 124.199} C_DIS
LIN {X 0.075,Y -315.810,Z 1468.690,A 0.000,B 0.000,C 90.000,E1 124.119} C_DIS
LIN {X 0.131,Y -319.887,Z 1468.688,A 0.000,B 0.000,C 90.000,E1 123.913} C_DIS
LIN {X 0.187,Y -322.281,Z 1468.688,A 0.000,B 0.000,C 90.000,E1 123.706} C_DIS
LIN {X 0.096,Y -326.105,Z 1468.685,A 0.000,B 0.000,C 90.000,E1 123.245} C_DIS
LIN {X -0.088,Y -327.867,Z 1468.683,A 0.000,B 0.000,C 90.000,E1 122.959} C_DIS
LIN {X -0.166,Y -330.381,Z 1468.679,A 0.000,B 0.000,C 90.000,E1 122.339} C_DIS
LIN {X 0.074,Y -341.276,Z 1468.664,A 0.000,B 0.000,C 90.000,E1 119.489} C_DIS
LIN {X 0.008,Y -353.542,Z 1468.649,A 0.000,B 0.000,C 90.000,E1 116.744} C_DIS
LIN {X 0.128,Y -367.291,Z 1468.634,A 0.000,B 0.000,C 90.000,E1 114.027} C_DIS
LIN {X -0.117,Y -380.848,Z 1468.621,A 0.000,B 0.000,C 90.000,E1 111.716} C_DIS
LIN {X 0.045,Y -395.763,Z 1468.608,A 0.000,B 0.000,C 90.000,E1 109.396} C_DIS
LIN {X -0.051,Y -412.137,Z 1468.595,A 0.000,B 0.000,C 90.000,E1 107.166} C_DIS
LIN {X 0.138,Y -430.086,Z 1468.583,A 0.000,B 0.000,C 90.000,E1 104.954} C_DIS
LIN {X -0.194,Y -449.589,Z 1468.571,A 0.000,B 0.000,C 90.000,E1 102.883} C_DIS
LIN {X 0.072,Y -469.822,Z 1468.561,A 0.000,B 0.000,C 90.000,E1 100.894} C_DIS
LIN {X 0.017,Y -487.932,Z 1468.552,A 0.000,B 0.000,C 90.000,E1 99.321} C_DIS
LIN {X 0.089,Y -490.096,Z 1468.551,A 0.000,B 0.000,C 90.000,E1 99.095} C_DIS
LIN {X 0.014,Y -491.912,Z 1468.549,A 0.000,B 0.000,C 90.000,E1 98.859} C_DIS
LIN {X -0.063,Y -493.276,Z 1468.548,A 0.000,B 0.000,C 90.000,E1 98.624} C_DIS
LIN {X 0.170,Y -495.000,Z 1468.545,A 0.000,B 0.000,C 90.000,E1 98.106} C_DIS
LIN {X -0.078,Y -495.625,Z 1468.542,A 0.000,B 0.000,C 90.000,E1 97.644} C_DIS
LIN {X 0.177,Y -495.254,Z 1468.540,A 0.000,B 0.000,C 90.000,E1 97.125} C_DIS
LIN {X -0.057,Y -493.836,Z 1468.537,A 0.000,B 0.000,C 90.000,E1 96.663} C_DIS
LIN {X -0.146,Y -492.660,Z 1468.536,A 0.000,B 0.000,C 90.000,E1 96.429} C_DIS
LIN {X 0.188,Y -479.561,Z 1468.525,A 0.000,B 0.000,C 90.000,E1 94.416} C_DIS
LIN {X 0.115,Y -470.482,Z 1468.516,A 0.000,B 0.000,C 90.000,E1 92.922} C_DIS
LIN {X -0.201,Y -464.102,Z 1468.511,A 0.000,B 0.000,C 90.000,E1 91.949} C_DIS
LIN {X -0.094,Y -453.990,Z 1468.502,A 0.000,B 0.000,C 90.000,E1 90.401} C_DIS
LIN {X -0.043,Y -438.646,Z 1468.489,A 0.000,B 0.000,C 90.000,E1 88.051} C_DIS
LIN {X 0.062,Y -428.466,Z 1468.480,A 0.000,B 0.000,C 90.000,E1 86.445} C_DIS
LIN {X 0.104,Y -416.530,Z 1468.470,A 0.000,B 0.000,C 90.000,E1 84.552} C_DIS
LIN {X -0.073,Y -406.285,Z 1468.461,A 0.000,B 0.000,C 90.000,E1 82.932} C_DIS
LIN {X 0.067,Y -392.403,Z 1468.448,A 0.000,B 0.000,C 90.000,E1 80.679} C_DIS
LIN {X 0.032,Y -375.411,Z 1468.432,A 0.000,B 0.000,C 90.000,E1 77.825} C_DIS
LIN {X 0.155,Y -362.364,Z 1468.419,A 0.000,B 0.000,C 90.000,E1 75.463} C_DIS
LIN {X 0.129,Y -351.077,Z 1468.408,A 0.000,B 0.000,C 90.000,E1 73.378} C_DIS
LIN {X -0.036,Y -339.702,Z 1468.396,A 0.000,B 0.000,C 90.000,E1 71.275} C_DIS
LIN {X 0.070,Y -326.972,Z 1468.382,A 0.000,B 0.000,C 90.000,E1 68.773} C_DIS
LIN {X 0.011,Y -310.419,Z 1468.363,A 0.000,B 0.000,C 90.000,E1 65.281} C_DIS
LIN {X -0.077,Y -296.401,Z 1468.344,A 0.000,B 0.000,C 90.000,E1 62.025} C_DIS
LIN {X -0.011,Y -284.742,Z 1468.328,A 0.000,B 0.000,C 90.000,E1 58.997} C_DIS
LIN {X -0.063,Y -273.704,Z 1468.311,A 0.000,B 0.000,C 90.000,E1 55.928} C_DIS
LIN {X 0.034,Y -263.085,Z 1468.293,A 0.000,B 0.000,C 90.000,E1 52.763} C_DIS
LIN {X 0.095,Y -253.063,Z 1468.275,A 0.000,B 0.000,C 90.000,E1 49.542} C_DIS
LIN {X -0.167,Y -242.827,Z 1468.255,A 0.000,B 0.000,C 90.000,E1 45.972} C_DIS
LIN {X -0.054,Y -233.585,Z 1468.235,A 0.000,B 0.000,C 90.000,E1 42.243} C_DIS
LIN {X -0.023,Y -225.408,Z 1468.214,A 0.000,B 0.000,C 90.000,E1 38.463} C_DIS
